// TwinCAT 3 PLC project PLC1
// ProgramVersion: 3.1.4026.24
// CompilerDefines: VISU_USEPROPERTYINFO
// libraries:
//   Tc2_Standard, * (Beckhoff Automation GmbH)
//   Tc2_System, * (Beckhoff Automation GmbH)
// project tree:
//   DUTs/ E_AutoStep.TcDUT, E_ControlMode.TcDUT (not stored), E_LogSev.TcDUT (not stored), E_MasterAutoStep.TcDUT, E_RobotConnState.TcDUT (not stored), ST_HmiMasterAuto.TcDUT, ST_HmiMasterAutoCfg.TcDUT, ST_HmiPiston.TcDUT, ST_HmiPistonAuto.TcDUT (not stored), ST_HmiPistonAutoCfg.TcDUT, ST_HmiRobot.TcDUT, ST_LogBridgeCfg.TcDUT (not stored), ST_LogEntry.TcDUT (not stored)
//   / GlobalTextList.TcGTLO, IOmapTask.TcTTO (not stored), PlcTask.TcTTO, Visualization Manager.TcVMO (not stored)
//   GVLs/ GVL_App.TcGVL, GVL_HMI.TcGVL, GVL_HmiPersistent.TcGVL, GVL_IO.TcGVL, GVL_Log.TcGVL, GVL_Robot.TcGVL (not stored)
//   POUs/ F_LogEvent.TcPOU, FB_MasterAutoCycle.TcPOU, FB_PistonAutoCycle.TcPOU, FB_SolSolPiston_2Pos.TcPOU, FB_SolSpringPiston_2Pos.TcPOU, MAIN.TcPOU, PRG_IoMap.TcPOU
//   VISUs/ VISU_Home.TcVIS, VISU_Piston.TcVIS, VISU_Pistons.TcVIS, VISU_Robot.TcVIS, VISU_AutoCycle.TcVIS, VISU_Diagnostics.TcVIS
// real-time tasks:
//   TASK PlcTask: cycle T#10ms, priority 20, ADS port 350
//   TASK IOmapTask: cycle T#5ms, priority 15, ADS port 351
// I/O:
//   DEVICE Device 1 (EtherCAT) (disabled), AmsNetId 192.168.1.101.2.1
//     Term 1 (EK1100) [EK1100 EtherCAT Coupler (2A E-Bus)]
//       Term 2 (EL2008) [EL2008 8Ch. Dig. Output 24V, 0.5A]
//       Term 3 (EL1008) [EL1008 8Ch. Dig. Input 24V, 3ms]
// variable links:
//   PLC1/PLC1 Instance <-> Device 1 (EtherCAT)/Term 1 (EK1100)/Term 2 (EL2008)
//     IOmapTask Outputs/GVL_IO.dOut[{1..8}] <-> Channel {1..8}/GVL_IO.dOut[{1..8}]  (8 links)
//   PLC1/PLC1 Instance <-> Device 1 (EtherCAT)/Term 1 (EK1100)/Term 3 (EL1008)
//     IOmapTask Inputs/GVL_IO.dIn[{1..8}] <-> Channel {1..8}/GVL_IO.dIn[{1..8}]  (8 links)

CONFIGURATION PLC1
    RESOURCE PLC ON TwinCAT3
        TASK PlcTask(INTERVAL := T#10ms, PRIORITY := 20);
        PROGRAM MAIN WITH PlcTask : MAIN;
    END_RESOURCE
END_CONFIGURATION

// ---- DUTs/E_AutoStep.TcDUT
{attribute 'qualified_only'}
{attribute 'strict'}
{attribute 'to_string'}
TYPE E_AutoStep :
(
    IDLE       := 0,
    EXTENDING  := 1,
    DWELL_EXT  := 2,
    RETRACTING := 3,
    DWELL_RET  := 4,
    ERR        := 99
) ;
END_TYPE

// ---- DUTs/E_MasterAutoStep.TcDUT
{attribute 'qualified_only'}
{attribute 'strict'}
{attribute 'to_string'}
TYPE E_MasterAutoStep :
(
    IDLE                 := 0,
    SEP_EXTENDING        := 1,
    WAIT_POS2            := 2,
    PUSH_EXTENDING       := 3,
    DWELL_PUSH           := 4,
    PUSH_RETRACTING      := 5,
    PUSH_RETRACTED_DWELL := 6,
    SEP_RETRACTING       := 7,
    SEP_RETRACTED_DWELL  := 8,
    INIT_PUSH_RETRACTING := 10,
    INIT_SEP_RETRACTING  := 11,
    INIT_GRIP_RETRACTING := 12,
    WAIT_PLATE           := 20,
    GRIP_EXTENDING       := 21,
    GRIP_RETRACTING      := 22,
    ERR                  := 99
) ;
END_TYPE

// ---- DUTs/ST_HmiMasterAuto.TcDUT
TYPE ST_HmiMasterAuto :
STRUCT
    // Display label ('MasterAuto'). Set from GVL_HMI init, never written by FB.
    Name             : STRING(30);

    // HMI writes -- momentary command buttons (R_TRIG inside FB latches the rising edge)
    bStart           : BOOL;
    bStop            : BOOL;
    bReset           : BOOL;

    // FB writes -- status
    eStep            : E_MasterAutoStep;
    sStepText        : STRING(20);   // human-readable mirror of eStep
    tElapsedS        : LREAL;        // seconds spent in the current step (0.0 on transition)
    iErrorCode       : INT;          // 0 = OK; see FB_MasterAutoCycle header for the code table
    sErrorText       : STRING(80);
    nCyclesCompleted : UDINT;        // incremented at end of GRIP_RETRACTING

    // HMI writes -- bench sim of the robot's start handshake. OR-ed with the
    // real stRobot.bStartAssembly level; FB auto-clears it after the rising
    // edge is consumed (never writes the robot-owned signal itself).
    bSimStartAssembly      : BOOL;

    // HMI writes -- per-step Simulate flags. Rising edge shortcuts the current
    // step's wait condition (FB clears the flag on consumption via R_TRIG.Q).
    bSimStep_Idle          : BOOL;
    bSimStep_InitPushRet   : BOOL;
    bSimStep_InitSepRet    : BOOL;
    bSimStep_InitGripRet   : BOOL;
    bSimStep_WaitPlate     : BOOL;
    bSimStep_GripExt       : BOOL;
    bSimStep_SepExt        : BOOL;
    bSimStep_WaitPos2      : BOOL;
    bSimStep_PushExt       : BOOL;
    bSimStep_DwellPush     : BOOL;
    bSimStep_PushRet       : BOOL;
    bSimStep_PushRetDwell  : BOOL;
    bSimStep_SepRet        : BOOL;
    bSimStep_SepRetDwell   : BOOL;
    bSimStep_GripRet       : BOOL;
END_STRUCT
END_TYPE

// ---- DUTs/ST_HmiMasterAutoCfg.TcDUT
TYPE ST_HmiMasterAutoCfg :
STRUCT
    // Timers, milliseconds. UDINT so HMI NumericInput binds directly.
    tDwellPushMs            : UDINT := 2000;   // DWELL_PUSH -- hold at push-extended
    tPushRetractedDwellMs   : UDINT := 500;    // PUSH_RETRACTED_DWELL -- hold after push retract
    tSepRetractedDwellMs    : UDINT := 500;    // SEP_RETRACTED_DWELL -- hold after sep retract before IDLE

    // Timeout guards every non-DWELL waiting state. On expiry, iErrorCode is
    // set to the step's numeric code and the cycle enters ERR.
    tStepTimeoutMs          : UDINT := 10000;

    // Dedicated timeout for WAIT_PLATE (bounded by robot placement time, not
    // by a motion budget). On expiry, iErrorCode := 9 and the cycle enters ERR.
    tPlateWaitTimeoutMs     : UDINT := 10000;

    // If TRUE, the 4 movement states ignore sensor feedback and advance when
    // tStepTimeoutMs expires — the timeout doubles as the fixed step duration.
    // No timeout-error path while sensorless. Mirrors ST_HmiPistonAutoCfg.bNoSensors.
    bNoSensors              : BOOL  := FALSE;

    // While TRUE, IDLE immediately starts the next cycle (no START or
    // robot CMD:1 edge needed). Uncheck to stop after the cycle returns
    // to IDLE. Cleared by the FB on entry to ERR so a RESET does not
    // instantly restart motion.
    bContinuous             : BOOL  := FALSE;

    // Global machine mode — single source of truth for every piston's mode.
    // BOOL so the classic VISU HMI (boolean-only) binds a checkbox directly,
    // matching the per-piston bMode convention. FALSE = Manual (operator jogs
    // each piston; master cycle held in IDLE). TRUE = Automatic (MasterAutoCycle
    // owns all six pistons). Enforced every scan in MAIN onto each piston's
    // eMode AND bMode, so there is no per-piston double-control.
    bAutoMode               : BOOL := FALSE;
END_STRUCT
END_TYPE

// ---- DUTs/ST_HmiPiston.TcDUT
TYPE ST_HmiPiston :
STRUCT
    // Display label ("Piston 1", "Ejector", ...). Set from GVL_HMI, never written by FB.
    Name               : STRING(30);

    // HMI writes — mode
    eMode              : E_ControlMode;
	bMode				: BOOL; // to be able to control from the VISU old HMI

    // HMI writes — latched command targets (momentary press, rising edge selects)
    bManCmdExtend      : BOOL;
    bManCmdRetract     : BOOL;

    // HMI writes — jog while held (TRUE while operator holds the JOG button)
    bManJogExtend      : BOOL;
    bManJogRetract     : BOOL;

    // HMI writes — simulate sensor inputs (OR-merged with real). Future Sim checkbox hook.
    bSimulateExtended  : BOOL;
    bSimulateRetracted : BOOL;

    // HMI reads (FB writes) — latched-target highlight
    bSelectedExtend    : BOOL;
    bSelectedRetract   : BOOL;

    // HMI reads (FB writes) — effective sensor = real OR simulate
    bIsExtended        : BOOL;
    bIsRetracted       : BOOL;
    bIsMoving          : BOOL;

    // HMI reads — physical solenoid coil states (FB mirrors them every cycle)
    bOutSolenoidExtend  : BOOL;
    bOutSolenoidRetract : BOOL;
END_STRUCT
END_TYPE

// ---- DUTs/ST_HmiPistonAutoCfg.TcDUT
TYPE ST_HmiPistonAutoCfg :
STRUCT
    // All times in milliseconds. UDINT so HMI NumericInput binds directly (no TIME<->UDINT juggling).

    // Dwell = how long to sit at the sensor before starting the reverse move.
    tDwellExtendedMs   : UDINT := 500;
    tDwellRetractedMs  : UDINT := 500;

    // Timeout = if we do not see the target sensor within this window, raise an error.
    tTimeoutExtendMs   : UDINT := 3000;
    tTimeoutRetractMs  : UDINT := 3000;

    // If TRUE, DWELL_RET loops back to EXTENDING instead of returning to IDLE.
    bContinuous        : BOOL  := FALSE;
END_STRUCT
END_TYPE

// ---- DUTs/ST_HmiRobot.TcDUT
TYPE ST_HmiRobot :
STRUCT
    // Display label ('Robot'). Set from GVL_Robot, never written by bridge.
    Name           : STRING(30);

    // Bridge writes — connection state (enum + string mirror for HMI text binding)
    eConnState     : E_RobotConnState;
    sConnStateText : STRING(20);

    // Bridge writes — latched "in position N" flags. Bridge holds the last-seen
    // position TRUE and clears the other two when a new POS frame arrives.
    bAtPos1        : BOOL;
    bAtPos2        : BOOL;
    bAtPos3        : BOOL;

    // Bridge writes — diagnostics
    nPacketsRx     : UDINT;
    sLastMessage   : STRING(80);

    // Outbound pulses — PLC (FB_MasterAutoCycle) writes TRUE for one cycle.
    // Bridge polls each on rising edge, sends the corresponding TCP frame,
    // then clears the flag. If the bridge is disconnected the flag stays
    // TRUE until reconnect; no queue, no lost pulses.
    bTxAutoStarted  : BOOL;
    bTxPushDone     : BOOL;
    bTxPistonsError : BOOL;

    // Inbound pulse — bridge writes TRUE on receiving a RESET_ERROR frame.
    // FB_MasterAutoCycle consumes on rising edge and clears the flag.
    bRxResetError   : BOOL;

    // Bridge writes — outbound diagnostics
    nPacketsTx      : UDINT;
    sLastTxMessage  : STRING(80);
END_STRUCT
END_TYPE

// ---- GVLs/GVL_App.TcGVL
{attribute 'qualified_only'}
// Cooked IO aliases. Bound to the raw GVL_IO.dIn[i]/dOut[i] hardware arrays
// in MAIN's read-inputs / write-outputs bookends. No AT %*: these are plain
// BOOLs the FBs consume — the actual hardware wiring lives in GVL_IO.
//
// Tag convention: <Device>Sol<N>  = single EXTEND coil (SOL-Spring).
// The mechanical spring returns the actuator when the coil is de-energised,
// so no per-actuator Retract alias exists. DI still has a Retracted sensor.
//
//   SepSolN : Pin separator N   (DI 1..6, DO 1..3)
//   PushSolN: Pin push N        (DI 7..12, DO 4..6)
//   GripSolL / GripSolR: side grip pistons that clamp the robot-placed plate
//                       (DI 14..17, DO 8..9)
//   PlateSenL / PlateSenR: plate-presence sensors gating cycle start
//                         (DI 18..19)
//   PbN / LedPbN: panel push buttons + status LEDs (DI 20..22, DO 10..12).
//                Behavior mode-gated -- see field comments below.
//
// DO layout:
//   dOut[1..3] = SepSolN Extend
//   dOut[4..6] = PushSolN Extend
//   dOut[7]    = free (was Robot bAssemblyRunning; retired, comms are TCP-only)
//   dOut[8..9] = GripSolL/R Extend
//   dOut[10..12] = PB1/2/3 LEDs (see Phase B)
//   dOut[13..16] = free
VAR_GLOBAL
    // SepSol1 (Pin separator 1) — DI 1..2, DO 1
    bSensorSepRetracted1  : BOOL;
    bSensorSepExtended1   : BOOL;
    bValveSepExtend1      : BOOL;

    // SepSol2 (Pin separator 2) — DI 3..4, DO 2
    bSensorSepRetracted2  : BOOL;
    bSensorSepExtended2   : BOOL;
    bValveSepExtend2      : BOOL;

    // SepSol3 (Pin separator 3) — DI 5..6, DO 3
    bSensorSepRetracted3  : BOOL;
    bSensorSepExtended3   : BOOL;
    bValveSepExtend3      : BOOL;

    // PushSol1 (Pin push 1) — DI 7..8, DO 4
    bSensorPushRetracted1 : BOOL;
    bSensorPushExtended1  : BOOL;
    bValvePushExtend1     : BOOL;

    // PushSol2 (Pin push 2) — DI 9..10, DO 5
    bSensorPushRetracted2 : BOOL;
    bSensorPushExtended2  : BOOL;
    bValvePushExtend2     : BOOL;

    // PushSol3 (Pin push 3) — DI 11..12, DO 6
    bSensorPushRetracted3 : BOOL;
    bSensorPushExtended3  : BOOL;
    bValvePushExtend3     : BOOL;

    // GripSolL (side grip, left) — DI 14..15, DO 8
    bSensorGripRetractedL : BOOL;
    bSensorGripExtendedL  : BOOL;
    bValveGripExtendL     : BOOL;

    // GripSolR (side grip, right) — DI 16..17, DO 9
    bSensorGripRetractedR : BOOL;
    bSensorGripExtendedR  : BOOL;
    bValveGripExtendR     : BOOL;

    // Plate-presence sensors — DI 18..19 (input only; no coil)
    bPlateSenL : BOOL;
    bPlateSenR : BOOL;

    // Panel push buttons + status LEDs — DI 20..22 / DO 10..12.
    // PB1 in Auto  = cycle-start bypass (bypass of robot's CMD:1).
    // PB1 in Manual = hold to extend both grip pistons.
    // PB2 in Manual = hold to extend all 3 SepSol pistons.
    // PB3 in Manual = hold to extend all 3 PushSol pistons.
    // LEDs mirror the corresponding PB press state (wiring diagnostic).
    bPb1     : BOOL;
    bPb2     : BOOL;
    bPb3     : BOOL;
    bLedPb1  : BOOL;
    bLedPb2  : BOOL;
    bLedPb3  : BOOL;
END_VAR

// ---- GVLs/GVL_HMI.TcGVL
{attribute 'qualified_only'}
{attribute 'TcHmiSymbol.AddSymbol'}
VAR_GLOBAL
    stSepSol1  : ST_HmiPiston := (Name := 'SepSol1');
    stSepSol2  : ST_HmiPiston := (Name := 'SepSol2');
    stSepSol3  : ST_HmiPiston := (Name := 'SepSol3');
    stPushSol1 : ST_HmiPiston := (Name := 'PushSol1');
    stPushSol2 : ST_HmiPiston := (Name := 'PushSol2');
    stPushSol3 : ST_HmiPiston := (Name := 'PushSol3');
    stGripSolL : ST_HmiPiston := (Name := 'GripSolL');
    stGripSolR : ST_HmiPiston := (Name := 'GripSolR');

    // Runtime state for the per-piston auto sequencers. Config for each
    // lives in the matching stXxxAutoCfg in GVL_HmiPersistent (PERSISTENT).
    stSepSol1Auto  : ST_HmiPistonAuto;
    stSepSol2Auto  : ST_HmiPistonAuto;
    stSepSol3Auto  : ST_HmiPistonAuto;
    stPushSol1Auto : ST_HmiPistonAuto;
    stPushSol2Auto : ST_HmiPistonAuto;
    stPushSol3Auto : ST_HmiPistonAuto;

    // Plate-presence sensors exposed to the HMI (indicator lamps on the
    // AutoCycle page). Mirror of GVL_App.bPlateSen* driven in MAIN.
    bPlateSenL : BOOL;
    bPlateSenR : BOOL;

    // Runtime state for the master (multi-piston + robot-coordinated) auto
    // sequence. Config for it lives in GVL_HmiPersistent.stMasterAutoCfg.
    stMasterAuto   : ST_HmiMasterAuto := (Name := 'MasterAuto');
END_VAR

// ---- GVLs/GVL_HmiPersistent.TcGVL
{attribute 'qualified_only'}
{attribute 'TcHmiSymbol.AddSymbol'}
VAR_GLOBAL PERSISTENT
    // Auto-cycle configuration. PERSISTENT so operator-tuned dwell / timeout
    // values survive an Activate Configuration + PLC restart. Values reset
    // to the struct defaults only on a full cold-boot reset.
    stSepSol1AutoCfg  : ST_HmiPistonAutoCfg;
    stPushSol1AutoCfg : ST_HmiPistonAutoCfg;

    // Config for the master (multi-piston + robot-coordinated) auto sequence.
    // See ST_HmiMasterAutoCfg for the tunable list; defaults land on cold-boot.
    stMasterAutoCfg   : ST_HmiMasterAutoCfg;
END_VAR

// ---- GVLs/GVL_IO.TcGVL
{attribute 'qualified_only'}
VAR_GLOBAL
	dOut AT%Q* :ARRAY[1..16]OF BOOL;
	dIn  AT%I* :ARRAY[1..24]OF BOOL;
END_VAR

// ---- GVLs/GVL_Log.TcGVL
{attribute 'qualified_only'}
{attribute 'TcHmiSymbol.AddSymbol'}
VAR_GLOBAL
    // Ring buffer of the most recent log entries the PLC has produced.
    // The Python bridge polls nWriteIdx via ADS and drains new slots.
    //   write slot at any moment = (nWriteIdx MOD 256)
    //   overflow detected when (nWriteIdx - lastReadIdx) > 256
    aLog       : ARRAY[0..255] OF ST_LogEntry;

    // Monotonic write counter (never wraps in practice — UDINT overflows
    // after 2^32 writes ≈ 4.3 billion, decades even at 1 kHz logging).
    nWriteIdx  : UDINT;

    // Runtime toggle for DEBUG severity. F_LogEvent drops DBG entries
    // when this is FALSE. Operator can flip it from the HMI without a
    // rebuild. HMI ToggleSwitch on the Robot page binds here.
    bDebugMode : BOOL := FALSE;
END_VAR

// ---- POUs/MAIN.TcPOU
PROGRAM MAIN
VAR
    fbSepSol1  : FB_SolSpringPiston_2Pos;
    fbSepSol2  : FB_SolSpringPiston_2Pos;
    fbSepSol3  : FB_SolSpringPiston_2Pos;
    fbPushSol1 : FB_SolSpringPiston_2Pos;
    fbPushSol2 : FB_SolSpringPiston_2Pos;
    fbPushSol3 : FB_SolSpringPiston_2Pos;

    // Per-piston auto-cycle sequencers. Each drives one piston's
    // bAutoCmdExtend / bAutoCmdRetract via its bCmdExtend / bCmdRetract,
    // OR-merged with fbMasterAutoCycle's output at each piston call site.
    fbSepSol1Auto  : FB_PistonAutoCycle;
    fbSepSol2Auto  : FB_PistonAutoCycle;
    fbSepSol3Auto  : FB_PistonAutoCycle;
    fbPushSol1Auto : FB_PistonAutoCycle;
    fbPushSol2Auto : FB_PistonAutoCycle;
    fbPushSol3Auto : FB_PistonAutoCycle;

    // Full-machine sequencer coordinating the 3 pairs of (SepSolN,
    // PushSolN) plus the robot handshake. Its command outputs
    // OR-merge with the per-piston auto FBs at each piston call site.
    fbMasterAutoCycle : FB_MasterAutoCycle;
END_VAR

(* ==========================================
   Master auto-cycle — coordinates the 3 pairs of (Sep,Push) pistons
   with the robot handshake. Called BEFORE the per-piston
   auto FBs and BEFORE the piston FBs so its bSepCmd* / bPushCmd*
   outputs feed forward this scan.
   Master reads bIs* from the piston stHmi structs — those carry the
   previous scan's values (100 µs lag, negligible for a physical
   machine).
   ========================================== *)
fbMasterAutoCycle.bSepIsExtended[1]   := GVL_HMI.stSepSol1.bIsExtended;
fbMasterAutoCycle.bSepIsExtended[2]   := GVL_HMI.stSepSol2.bIsExtended;
fbMasterAutoCycle.bSepIsExtended[3]   := GVL_HMI.stSepSol3.bIsExtended;
fbMasterAutoCycle.bSepIsRetracted[1]  := GVL_HMI.stSepSol1.bIsRetracted;
fbMasterAutoCycle.bSepIsRetracted[2]  := GVL_HMI.stSepSol2.bIsRetracted;
fbMasterAutoCycle.bSepIsRetracted[3]  := GVL_HMI.stSepSol3.bIsRetracted;
fbMasterAutoCycle.bPushIsExtended[1]  := GVL_HMI.stPushSol1.bIsExtended;
fbMasterAutoCycle.bPushIsExtended[2]  := GVL_HMI.stPushSol2.bIsExtended;
fbMasterAutoCycle.bPushIsExtended[3]  := GVL_HMI.stPushSol3.bIsExtended;
fbMasterAutoCycle.bPushIsRetracted[1] := GVL_HMI.stPushSol1.bIsRetracted;
fbMasterAutoCycle.bPushIsRetracted[2] := GVL_HMI.stPushSol2.bIsRetracted;
fbMasterAutoCycle.bPushIsRetracted[3] := GVL_HMI.stPushSol3.bIsRetracted;
fbMasterAutoCycle(
    bStartAssembly := GVL_Robot.stRobot.bStartAssembly,
    stHmi          := GVL_HMI.stMasterAuto,
    stCfg          := GVL_HmiPersistent.stMasterAutoCfg,
    stRobot        := GVL_Robot.stRobot
);

(* Optional "Put all to Auto" mode: while the master cycle is running,
   force all six pistons into Automatic so bAutoCmd* reaches the coil.
   Gated by stMasterAutoCfg.bForceAllAuto — when FALSE (default), only
   pistons the operator explicitly put into Automatic participate in the
   master cycle. On IDLE / ERR this block does nothing, regardless of
   the flag. *)
IF fbMasterAutoCycle.bAnyRunning AND GVL_HmiPersistent.stMasterAutoCfg.bForceAllAuto THEN
    GVL_HMI.stSepSol1.eMode  := E_ControlMode.Automatic;
    GVL_HMI.stPushSol1.eMode := E_ControlMode.Automatic;
    GVL_HMI.stSepSol2.eMode  := E_ControlMode.Automatic;
    GVL_HMI.stPushSol2.eMode := E_ControlMode.Automatic;
    GVL_HMI.stSepSol3.eMode  := E_ControlMode.Automatic;
    GVL_HMI.stPushSol3.eMode := E_ControlMode.Automatic;
END_IF;

(* ==========================================
   Pin separators (SOL-Spring, 2 limit switches, single Extend coil).
   SepSol1 and PushSol1 are driven by their own FB_PistonAutoCycle
   instances (called first so their outputs feed the piston FB this
   cycle). All six pistons OR-merge with fbMasterAutoCycle's outputs
   so the master sequence can command any/all of them in parallel.
   ========================================== *)
fbSepSol1Auto(
    sName        := 'SepSol1Auto',
    stHmi        := GVL_HMI.stSepSol1,
    stAuto       := GVL_HMI.stSepSol1Auto,
    stCfg        := GVL_HmiPersistent.stSepSol1AutoCfg
    // bCmdExtend / bCmdRetract wired inline in the fbSepSol1 call below
);

fbSepSol1(
    bAutoCmdExtend   := fbSepSol1Auto.bCmdExtend  OR fbMasterAutoCycle.bSepCmdExtend[1],
    bAutoCmdRetract  := fbSepSol1Auto.bCmdRetract OR fbMasterAutoCycle.bSepCmdRetract[1],
    bSwitchExtended  := GVL_App.bSensorSepExtended1,
    bSwitchRetracted := GVL_App.bSensorSepRetracted1,
    stHmi            := GVL_HMI.stSepSol1,
    bOutSolenoid     => GVL_App.bValveSepExtend1
);

fbSepSol2Auto(
    sName        := 'SepSol2Auto',
    stHmi        := GVL_HMI.stSepSol2,
    stAuto       := GVL_HMI.stSepSol2Auto,
    stCfg        := GVL_HmiPersistent.stSepSol2AutoCfg
);

fbSepSol2(
    bAutoCmdExtend   := fbSepSol2Auto.bCmdExtend  OR fbMasterAutoCycle.bSepCmdExtend[2],
    bAutoCmdRetract  := fbSepSol2Auto.bCmdRetract OR fbMasterAutoCycle.bSepCmdRetract[2],
    bSwitchExtended  := GVL_App.bSensorSepExtended2,
    bSwitchRetracted := GVL_App.bSensorSepRetracted2,
    stHmi            := GVL_HMI.stSepSol2,
    bOutSolenoid     => GVL_App.bValveSepExtend2
);

fbSepSol3Auto(
    sName        := 'SepSol3Auto',
    stHmi        := GVL_HMI.stSepSol3,
    stAuto       := GVL_HMI.stSepSol3Auto,
    stCfg        := GVL_HmiPersistent.stSepSol3AutoCfg
);

fbSepSol3(
    bAutoCmdExtend   := fbSepSol3Auto.bCmdExtend  OR fbMasterAutoCycle.bSepCmdExtend[3],
    bAutoCmdRetract  := fbSepSol3Auto.bCmdRetract OR fbMasterAutoCycle.bSepCmdRetract[3],
    bSwitchExtended  := GVL_App.bSensorSepExtended3,
    bSwitchRetracted := GVL_App.bSensorSepRetracted3,
    stHmi            := GVL_HMI.stSepSol3,
    bOutSolenoid     => GVL_App.bValveSepExtend3
);

(* ==========================================
   Pin pushers
   ========================================== *)
fbPushSol1Auto(
    sName        := 'PushSol1Auto',
    stHmi        := GVL_HMI.stPushSol1,
    stAuto       := GVL_HMI.stPushSol1Auto,
    stCfg        := GVL_HmiPersistent.stPushSol1AutoCfg
    // bCmdExtend / bCmdRetract wired inline in the fbPushSol1 call below
);

fbPushSol1(
    bAutoCmdExtend   := fbPushSol1Auto.bCmdExtend  OR fbMasterAutoCycle.bPushCmdExtend[1],
    bAutoCmdRetract  := fbPushSol1Auto.bCmdRetract OR fbMasterAutoCycle.bPushCmdRetract[1],
    bSwitchExtended  := GVL_App.bSensorPushExtended1,
    bSwitchRetracted := GVL_App.bSensorPushRetracted1,
    stHmi            := GVL_HMI.stPushSol1,
    bOutSolenoid     => GVL_App.bValvePushExtend1
);

fbPushSol2Auto(
    sName        := 'PushSol2Auto',
    stHmi        := GVL_HMI.stPushSol2,
    stAuto       := GVL_HMI.stPushSol2Auto,
    stCfg        := GVL_HmiPersistent.stPushSol2AutoCfg
);

fbPushSol2(
    bAutoCmdExtend   := fbPushSol2Auto.bCmdExtend  OR fbMasterAutoCycle.bPushCmdExtend[2],
    bAutoCmdRetract  := fbPushSol2Auto.bCmdRetract OR fbMasterAutoCycle.bPushCmdRetract[2],
    bSwitchExtended  := GVL_App.bSensorPushExtended2,
    bSwitchRetracted := GVL_App.bSensorPushRetracted2,
    stHmi            := GVL_HMI.stPushSol2,
    bOutSolenoid     => GVL_App.bValvePushExtend2
);

fbPushSol3Auto(
    sName        := 'PushSol3Auto',
    stHmi        := GVL_HMI.stPushSol3,
    stAuto       := GVL_HMI.stPushSol3Auto,
    stCfg        := GVL_HmiPersistent.stPushSol3AutoCfg
);

fbPushSol3(
    bAutoCmdExtend   := fbPushSol3Auto.bCmdExtend  OR fbMasterAutoCycle.bPushCmdExtend[3],
    bAutoCmdRetract  := fbPushSol3Auto.bCmdRetract OR fbMasterAutoCycle.bPushCmdRetract[3],
    bSwitchExtended  := GVL_App.bSensorPushExtended3,
    bSwitchRetracted := GVL_App.bSensorPushRetracted3,
    stHmi            := GVL_HMI.stPushSol3,
    bOutSolenoid     => GVL_App.bValvePushExtend3
);

END_PROGRAM

// ---- POUs/FB_SolSpringPiston_2Pos.TcPOU
FUNCTION_BLOCK FB_SolSpringPiston_2Pos
(* Single-solenoid, spring-return 2-position actuator.
   Coil energised  -> drives to EXTENDED.
   Coil de-energised -> mechanical spring returns to RETRACTED.

   The coil is a continuous force against the spring, so Section 2 uses a
   LATCH-and-RETAIN pattern: the coil is set TRUE on Extend command and
   FALSE on Retract command, and RETAINS its state (via VAR_OUTPUT retain)
   any cycle no explicit command is active. Without the latch the coil
   would drop the moment the extended sensor fires and the spring would
   immediately pull the piston back.

   Fail-safe by construction: broken wire, dead coil, PLC power loss
   or e-stop all leave bOutSolenoid FALSE and the spring retracts.

   Interface is kept symmetric with FB_SolSolPiston_2Pos so a sequencer FB
   (e.g. FB_PistonAutoCycle) can drive either actuator type without a
   custom variant. Reuses ST_HmiPiston unchanged; the retract-coil mirror
   field (stHmi.bOutSolenoidRetract) is always FALSE because no retract
   coil exists on this actuator. *)
VAR_INPUT
    (* Automatic Commands from PLC sequence logic. Wired to FALSE in MAIN until FB_Auto exists. *)
    bAutoCmdExtend    : BOOL;
    bAutoCmdRetract   : BOOL;

    (* External jog request (e.g. panel push-button). OR-merged with the
       HMI's stHmi.bManJogExtend inside so a physical PB and the HMI
       button can drive the same jog without stepping on each other.
       Only takes effect while eMode = Manual (same gate as the HMI jog). *)
    bJogExtend        : BOOL;

    (* Physical Feedback (Proximity Switches) *)
    bSwitchExtended   : BOOL;
    bSwitchRetracted  : BOOL;
END_VAR

VAR_IN_OUT
    (* HMI contract — mode, manual + simulate inputs, latched + sensor status *)
    stHmi             : ST_HmiPiston;
END_VAR

VAR_OUTPUT
    (* Physical Output to Solenoid — SINGLE coil.
       TRUE  = coil energised, actuator drives EXTENDED.
       FALSE = coil de-energised, spring returns actuator to RETRACTED. *)
    bOutSolenoid      : BOOL;
END_VAR

VAR
    (* Internal Target States *)
    bTargetExtend     : BOOL;
    bTargetRetract    : BOOL;

    (* HMI Manual-Button Edge Detection *)
    fbTrigManExtend   : R_TRIG;
    fbTrigManRetract  : R_TRIG;

    (* Effective sensor states = real OR HMI simulate. Recomputed every cycle in Section 0a. *)
    bSwitchExtended_eff  : BOOL;
    bSwitchRetracted_eff : BOOL;

    (* Previous-cycle snapshots for the mode-field bridge in Section 0b.
       Classic PLC HMI writes stHmi.bMode (Rotary Switch is boolean-only);
       web HMI writes stHmi.eMode (enum via ToggleSwitch). This FB is the
       authoritative reader of eMode, so we sync in whichever direction
       changed since last cycle. *)
    bPrevMode : BOOL;
    ePrevMode : E_ControlMode;
END_VAR

(* ==========================================
   0b. MODE-FIELD BRIDGE — sync bMode <-> eMode
   The classic PLC HMI (VISUs) writes stHmi.bMode because its Rotary Switch
   element is boolean-only. The web HMI (Flower_HMI) writes stHmi.eMode via
   a ToggleSwitch. Rest of this FB reads eMode as the authoritative field,
   so we mirror bMode into eMode when the classic HMI toggled the switch,
   and mirror eMode back into bMode when the web HMI (or anyone else) wrote
   eMode. Edge-triggered — whichever side changed since last cycle wins.
   Runs BEFORE Section 0 so downstream logic sees a coherent eMode.
   ========================================== *)
IF stHmi.bMode <> bPrevMode THEN
    // Classic VISU changed bMode → propagate to eMode
    IF stHmi.bMode THEN
        stHmi.eMode := E_ControlMode.Automatic;
    ELSE
        stHmi.eMode := E_ControlMode.Manual;
    END_IF;
ELSIF stHmi.eMode <> ePrevMode THEN
    // Web HMI (or any other writer) changed eMode → propagate to bMode
    stHmi.bMode := (stHmi.eMode = E_ControlMode.Automatic);
END_IF;

bPrevMode := stHmi.bMode;
ePrevMode := stHmi.eMode;

(* ==========================================
   0a. EFFECTIVE SENSOR INPUTS (real OR HMI simulate)
   ========================================== *)
bSwitchExtended_eff  := bSwitchExtended  OR stHmi.bSimulateExtended;
bSwitchRetracted_eff := bSwitchRetracted OR stHmi.bSimulateRetracted;

(* ==========================================
   0. HMI MANUAL BUTTON LATCHING (Radio-Button Behavior)
   ========================================== *)
fbTrigManExtend(CLK := stHmi.bManCmdExtend);
fbTrigManRetract(CLK := stHmi.bManCmdRetract);

// Independent IFs (not ELSIF): if multiple edges fire in the same cycle, the last one wins (Retract > Extend).
IF fbTrigManExtend.Q  THEN stHmi.bSelectedExtend := TRUE;  stHmi.bSelectedRetract := FALSE; END_IF;
IF fbTrigManRetract.Q THEN stHmi.bSelectedExtend := FALSE; stHmi.bSelectedRetract := TRUE;  END_IF;

IF stHmi.eMode = E_ControlMode.Automatic THEN
    stHmi.bSelectedExtend := FALSE; stHmi.bSelectedRetract := FALSE;
END_IF;

(* ==========================================
   1. MODE SELECTION & COMMAND MAPPING
   Spring-return semantics: both bAutoCmd* inputs are accepted for interface
   parity with FB_SolSolPiston_2Pos, but physically only Extend commands the
   coil. If both auto bits are TRUE we treat it as a conflict and de-energise
   (safe default — spring retracts).
   ========================================== *)
IF stHmi.eMode = E_ControlMode.Automatic THEN
    bTargetExtend  := bAutoCmdExtend  AND NOT bAutoCmdRetract;
    bTargetRetract := bAutoCmdRetract AND NOT bAutoCmdExtend;

ELSIF stHmi.eMode = E_ControlMode.Manual THEN
    bTargetExtend  := stHmi.bSelectedExtend;
    bTargetRetract := stHmi.bSelectedRetract;

ELSE
    // Safe default: undefined mode → no targets
    bTargetExtend  := FALSE;
    bTargetRetract := FALSE;
END_IF;

(* ==========================================
   1a. JOG OVERRIDE — clear latched selection while either jog is held
   ========================================== *)
// Section 1 above already copied stHmi.bSelected* into bTarget*. The stale
// bTarget* is harmless because Section 2's jog branches sit ahead of the
// bTarget* branches in the IF/ELSIF ladder and preempt them.
IF stHmi.bManJogExtend OR stHmi.bManJogRetract OR bJogExtend THEN
    stHmi.bSelectedExtend := FALSE; stHmi.bSelectedRetract := FALSE;
END_IF;

(* ==========================================
   1b. TARGET-REACHED RESET — clear bSelected* once the piston arrives
   ========================================== *)
IF stHmi.bSelectedExtend  AND bSwitchExtended_eff  THEN stHmi.bSelectedExtend  := FALSE; END_IF;
IF stHmi.bSelectedRetract AND bSwitchRetracted_eff THEN stHmi.bSelectedRetract := FALSE; END_IF;

(* ==========================================
   2. SOLENOID CONTROL — single coil, LATCH-and-RETAIN
   The coil is a continuous force against the spring. If it drops, the spring
   wins and the actuator retracts. So the coil must be LATCHED TRUE from the
   moment Extend is commanded until Retract is commanded — not pulsed until
   the sensor fires (which is the double-solenoid pattern).
   Structure:
     - Jog branches first, gated by Manual mode.
     - Explicit Extend / Retract command branches drive the coil to a
       definite state.
     - The IF ladder has NO ELSE. When no branch matches, VAR_OUTPUT retain
       semantics carry the coil forward:
         * At the Extended sensor after a successful extend (Section 1b just
           cleared bTargetExtend) → coil retains TRUE → piston HOLDS.
         * At the Retracted sensor after a successful retract → coil retains
           FALSE → piston HOLDS retracted (spring already there).
         * Sequencer DWELL_EXT (both auto bits FALSE) → coil retains TRUE
           for the full dwell instead of releasing the piston.
     - No sensor guards on the drive branches: holding the coil TRUE while
       at the Extended sensor is normal operation, not a wasted drive.
   Fail-safe still holds: cold boot, PLC reset, or e-stop leave bOutSolenoid
   at its default FALSE and the spring retracts.
   ========================================== *)
// JOG EXTEND: while held in Manual, energise coil. HMI-owned bManJogExtend
// OR external bJogExtend (panel push-button) -- both share the Manual gate.
IF (stHmi.bManJogExtend OR bJogExtend) AND stHmi.eMode = E_ControlMode.Manual THEN
    bOutSolenoid := TRUE;

// JOG RETRACT: while held in Manual, de-energise coil (spring retracts)
ELSIF stHmi.bManJogRetract AND stHmi.eMode = E_ControlMode.Manual THEN
    bOutSolenoid := FALSE;

// EXTEND commanded — energise coil (latched via retain when bTargetExtend clears)
ELSIF bTargetExtend THEN
    bOutSolenoid := TRUE;

// RETRACT commanded — de-energise coil, spring retracts
ELSIF bTargetRetract THEN
    bOutSolenoid := FALSE;

// No branch → bOutSolenoid RETAINS its previous value (see block header).
END_IF;

(* ==========================================
   3. HMI STATUS FEEDBACK
   bIsMoving is derived from sensor state alone: with Section 2's latch
   semantics, bOutSolenoid stays TRUE at the extended limit — so ORing
   it in would report "moving" while the piston is actually parked.
   "Between the two limits" is accurate for both strokes: coil-driven
   extend and spring-driven retract both traverse that gap.

   bOutSolenoidRetract is written FALSE unconditionally — no retract coil
   exists on a spring-return actuator, so the mirror stays cleared.
   ========================================== *)
stHmi.bIsExtended         := bSwitchExtended_eff;
stHmi.bIsRetracted        := bSwitchRetracted_eff;
stHmi.bIsMoving           := NOT bSwitchExtended_eff AND NOT bSwitchRetracted_eff;
stHmi.bOutSolenoidExtend  := bOutSolenoid;
stHmi.bOutSolenoidRetract := FALSE;

END_FUNCTION_BLOCK

// ---- POUs/FB_PistonAutoCycle.TcPOU
FUNCTION_BLOCK FB_PistonAutoCycle
VAR_INPUT
    (* Instance name used as the log source (e.g. 'SepSol1Auto').
       Kept as VAR_INPUT so the FB is reusable across pistons — MAIN passes
       the actual name at each call site. *)
    sName : STRING(20);
END_VAR

VAR_IN_OUT
    (* Reads bIs* effective sensors, writes eMode := Automatic while running. *)
    stHmi  : ST_HmiPiston;
    (* Reads commands, writes step + status. *)
    stAuto : ST_HmiPistonAuto;
    (* Reads persistent dwell / timeout / continuous config. *)
    stCfg  : ST_HmiPistonAutoCfg;
END_VAR

VAR_OUTPUT
    (* Wire these to the piston FB's bAutoCmdExtend / bAutoCmdRetract in MAIN. *)
    bCmdExtend  : BOOL;
    bCmdRetract : BOOL;
END_VAR

VAR
    (* HMI button edge detection *)
    fbTrigStart : R_TRIG;
    fbTrigStop  : R_TRIG;
    fbTrigReset : R_TRIG;
    fbTrigAck   : R_TRIG;

    (* Per-state timers. TON.IN bound to (eStep = target); .Q fires when PT elapsed.
       When we transition out, IN goes FALSE and TON auto-resets ET. *)
    fbTimerExtend  : TON;   // extend-timeout (fault on Q while EXTENDING)
    fbTimerRetract : TON;   // retract-timeout (fault on Q while RETRACTING)
    fbTimerDwellE  : TON;   // dwell at extended
    fbTimerDwellR  : TON;   // dwell at retracted

    (* Step-elapsed display timer. Resets on step change; long PT so .Q never fires. *)
    fbStepTimer : TON;

    (* Prev-state snapshot for step-changed detection *)
    ePrevStep    : E_AutoStep;
    bStepChanged : BOOL;
END_VAR

(* ==========================================
   0. HMI COMMAND EDGE DETECTION
   ========================================== *)
fbTrigStart(CLK := stAuto.bStart);
fbTrigStop (CLK := stAuto.bStop);
fbTrigReset(CLK := stAuto.bReset);
fbTrigAck  (CLK := stAuto.bAck);

(* ==========================================
   1. PER-STATE TIMERS
   Called BEFORE the state machine so their .Q outputs reflect the current
   state's dwell / timeout for this cycle's decisions.
   ========================================== *)
fbTimerExtend (IN := stAuto.eStep = E_AutoStep.EXTENDING,  PT := UDINT_TO_TIME(stCfg.tTimeoutExtendMs));
fbTimerRetract(IN := stAuto.eStep = E_AutoStep.RETRACTING, PT := UDINT_TO_TIME(stCfg.tTimeoutRetractMs));
fbTimerDwellE (IN := stAuto.eStep = E_AutoStep.DWELL_EXT,  PT := UDINT_TO_TIME(stCfg.tDwellExtendedMs));
fbTimerDwellR (IN := stAuto.eStep = E_AutoStep.DWELL_RET,  PT := UDINT_TO_TIME(stCfg.tDwellRetractedMs));

(* ==========================================
   2. GLOBAL COMMANDS
   Stop = soft interrupt back to IDLE (does NOT clear error latch).
   Reset = hard reset: force IDLE, clear cycles + error.
   Ack = clear error latch (only meaningful from ERR).
   ========================================== *)
IF fbTrigStop.Q AND stAuto.eStep <> E_AutoStep.ERR THEN
    stAuto.eStep := E_AutoStep.IDLE;
END_IF

IF fbTrigReset.Q THEN
    stAuto.eStep            := E_AutoStep.IDLE;
    stAuto.bError           := FALSE;
    stAuto.sErrorText       := '';
    stAuto.nCyclesCompleted := 0;
END_IF

IF fbTrigAck.Q AND stAuto.eStep = E_AutoStep.ERR THEN
    stAuto.bError     := FALSE;
    stAuto.sErrorText := '';
    stAuto.eStep      := E_AutoStep.IDLE;
END_IF

(* ==========================================
   3. STATE MACHINE
   Reads effective sensors from stHmi.bIsExtended / bIsRetracted — these
   are already the real-OR-simulate value written by the piston FB
   (FB_SolSolPiston_2Pos or FB_SolSpringPiston_2Pos). So simulation
   "just works" via the piston FB's existing bSimulate* pins.
   ========================================== *)
CASE stAuto.eStep OF

    E_AutoStep.IDLE:
        bCmdExtend  := FALSE;
        bCmdRetract := FALSE;
        (* Start only from IDLE (and only if no latched error). *)
        IF fbTrigStart.Q AND NOT stAuto.bError THEN
            stAuto.eStep := E_AutoStep.EXTENDING;
        END_IF

    E_AutoStep.EXTENDING:
        bCmdExtend  := TRUE;
        bCmdRetract := FALSE;
        stHmi.eMode := E_ControlMode.Automatic;
        IF stCfg.bNoSensors THEN
            (* Sensorless: PT = extend duration; timer expiry = success. *)
            IF fbTimerExtend.Q THEN
                stAuto.eStep := E_AutoStep.DWELL_EXT;
            END_IF
        ELSE
            (* Feedback mismatch = physical impossibility, sensor fault. *)
            IF stHmi.bIsExtended AND stHmi.bIsRetracted THEN
                stAuto.bError     := TRUE;
                stAuto.sErrorText := 'Both sensors active during EXTENDING (feedback mismatch)';
                stAuto.eStep      := E_AutoStep.ERR;
            ELSIF stHmi.bIsExtended THEN
                stAuto.eStep := E_AutoStep.DWELL_EXT;
            ELSIF fbTimerExtend.Q THEN
                stAuto.bError     := TRUE;
                stAuto.sErrorText := 'Timeout waiting for extended sensor';
                stAuto.eStep      := E_AutoStep.ERR;
            END_IF
        END_IF

    E_AutoStep.DWELL_EXT:
        (* Coil released — piston sits at the extended end sensor. *)
        bCmdExtend  := FALSE;
        bCmdRetract := FALSE;
        stHmi.eMode := E_ControlMode.Automatic;
        IF fbTimerDwellE.Q THEN
            stAuto.eStep := E_AutoStep.RETRACTING;
        END_IF

    E_AutoStep.RETRACTING:
        bCmdExtend  := FALSE;
        bCmdRetract := TRUE;
        stHmi.eMode := E_ControlMode.Automatic;
        IF stCfg.bNoSensors THEN
            (* Sensorless: PT = retract duration; timer expiry = success. *)
            IF fbTimerRetract.Q THEN
                stAuto.eStep := E_AutoStep.DWELL_RET;
            END_IF
        ELSE
            IF stHmi.bIsExtended AND stHmi.bIsRetracted THEN
                stAuto.bError     := TRUE;
                stAuto.sErrorText := 'Both sensors active during RETRACTING (feedback mismatch)';
                stAuto.eStep      := E_AutoStep.ERR;
            ELSIF stHmi.bIsRetracted THEN
                stAuto.eStep := E_AutoStep.DWELL_RET;
            ELSIF fbTimerRetract.Q THEN
                stAuto.bError     := TRUE;
                stAuto.sErrorText := 'Timeout waiting for retracted sensor';
                stAuto.eStep      := E_AutoStep.ERR;
            END_IF
        END_IF

    E_AutoStep.DWELL_RET:
        bCmdExtend  := FALSE;
        bCmdRetract := FALSE;
        stHmi.eMode := E_ControlMode.Automatic;
        IF fbTimerDwellR.Q THEN
            (* One complete cycle just ended. Count it. *)
            stAuto.nCyclesCompleted := stAuto.nCyclesCompleted + 1;
            IF stCfg.bContinuous THEN
                stAuto.eStep := E_AutoStep.EXTENDING;
            ELSE
                stAuto.eStep := E_AutoStep.IDLE;
            END_IF
        END_IF

    E_AutoStep.ERR:
        (* Latched error — outputs safe, wait for Ack or Reset. *)
        bCmdExtend  := FALSE;
        bCmdRetract := FALSE;
        (* Do NOT touch stHmi.eMode — let the operator flip to Manual for recovery. *)

END_CASE

(* ==========================================
   4. STEP-CHANGE DETECTION, LOGGING & ELAPSED TIMER
   Placed AFTER the state machine so we detect this cycle's transitions.
   fbStepTimer.IN := NOT bStepChanged pulses its ET back to 0 for one cycle
   on transition, then counts up until the next transition.
   ========================================== *)
bStepChanged := (stAuto.eStep <> ePrevStep);

(* Log every transition. ERR entries carry the human-readable sErrorText;
   all other transitions produce "PREV -> NEW" (relies on E_AutoStep's
   'to_string' attribute for label lookup). Runs AFTER bStepChanged is set
   but BEFORE ePrevStep is overwritten so we still have both endpoints. *)
IF bStepChanged THEN
    IF stAuto.eStep = E_AutoStep.ERR THEN
        F_LogEvent(eSev := E_LogSev.ERR, sSource := sName, sMsg := stAuto.sErrorText);
    ELSE
        F_LogEvent(
            eSev    := E_LogSev.INFO,
            sSource := sName,
            sMsg    := CONCAT(CONCAT(TO_STRING(ePrevStep), ' -> '), TO_STRING(stAuto.eStep))
        );
    END_IF
END_IF

ePrevStep := stAuto.eStep;

fbStepTimer(IN := NOT bStepChanged, PT := T#1D);
stAuto.tElapsedS := DINT_TO_LREAL(TIME_TO_DINT(fbStepTimer.ET)) * 0.001;

(* ==========================================
   5. STATUS TEXT MIRROR — refresh sStepText every cycle
   ========================================== *)
CASE stAuto.eStep OF
    E_AutoStep.IDLE:       stAuto.sStepText := 'Idle';
    E_AutoStep.EXTENDING:  stAuto.sStepText := 'Extending';
    E_AutoStep.DWELL_EXT:  stAuto.sStepText := 'Dwell (extended)';
    E_AutoStep.RETRACTING: stAuto.sStepText := 'Retracting';
    E_AutoStep.DWELL_RET:  stAuto.sStepText := 'Dwell (retracted)';
    E_AutoStep.ERR:        stAuto.sStepText := 'ERROR';
ELSE
    stAuto.sStepText := 'Unknown';
END_CASE

END_FUNCTION_BLOCK

// ---- POUs/F_LogEvent.TcPOU
(*
    Push one entry into the GVL_Log ring buffer.

    Callable from any scan without side effects on control logic. DEBUG entries
    are dropped when GVL_Log.bDebugMode = FALSE, so leaving DBG calls in
    production code costs nothing.

    Returns TRUE if the entry was recorded, FALSE if dropped by the debug filter.
*)
FUNCTION F_LogEvent : BOOL
VAR_INPUT
    eSev    : E_LogSev;
    sSource : STRING(20);
    sMsg    : STRING(80);
END_VAR
VAR
    idx : UDINT;
    k   : INT;
END_VAR

// Global mute — operator can disable ALL PLC logging from the HMI. When
// FALSE, we drop the event silently; the ring buffer and aRecent mirror
// are not touched so the last-known state stays visible.
IF NOT GVL_Log.bLogEnabled THEN
    F_LogEvent := FALSE;
    RETURN;
END_IF

// Debug filter — drop DBG severity when debug mode is off
IF (eSev = E_LogSev.DBG) AND NOT GVL_Log.bDebugMode THEN
    F_LogEvent := FALSE;
    RETURN;
END_IF

// Write into the ring at slot = nWriteIdx MOD 256
idx := GVL_Log.nWriteIdx MOD 256;
GVL_Log.aLog[idx].eSev    := eSev;
GVL_Log.aLog[idx].sSource := sSource;
GVL_Log.aLog[idx].sMsg    := sMsg;

// Shift the newest-first mirror down by one and write the new entry at
// [0]. HMI Logs page binds aRecent[0..19] directly in display order.
FOR k := 19 TO 1 BY -1 DO
    GVL_Log.aRecent[k] := GVL_Log.aRecent[k-1];
END_FOR
GVL_Log.aRecent[0].eSev    := eSev;
GVL_Log.aRecent[0].sSource := sSource;
GVL_Log.aRecent[0].sMsg    := sMsg;

// Increment the monotonic write counter — Python bridge polls this and
// drains any slots between its lastReadIdx and this value.
GVL_Log.nWriteIdx := GVL_Log.nWriteIdx + 1;

F_LogEvent := TRUE;

END_FUNCTION

// ---- POUs/FB_MasterAutoCycle.TcPOU
FUNCTION_BLOCK FB_MasterAutoCycle
(* Full-machine coordinated auto sequence spanning the robot and the 3
   pairs of SepSol / PushSol pistons (pair count fixed at 3 for this
   machine).

   Robot interface (TCP-only, 2026-07-26). The former discrete-I/O handshake
   is retired. All robot-side signals travel over FB_RobotTcpClient's
   STATE:n / CMD:n protocol:

     Robot -> PLC   nRobotCmd in {1,2}  (1=start, 2=reset error)
                    MAIN R_TRIGs on the edges; start pulse arrives here as
                    the VAR_INPUT bExtStartPulse.
     PLC -> Robot   nStateOut = TO_INT(eStep) or MANUAL(30)
                    Written by MAIN each scan, pushed by FB_RobotTcpClient
                    on change and as keep-alive.

   The cycle starts on any rising edge of bExtStartPulse (robot cmd=1, one
   scan wide), the HMI START button, or the sim-start flag.

   Sequence (all 3 Sep/Push pairs move in parallel; both grips move together):

     IDLE                    START button OR bExtStartPulse pulse OR SimIdle
                             OR bContinuous checked (level - keeps re-arming)
     INIT_PUSH_RETRACTING    drive PushCmdRetract[1..3]; wait AND of all
                             PushIsRetracted. Guarantees pistons are home before
                             a cycle starts, even if a prior manual move left
                             them extended.
     INIT_SEP_RETRACTING     drive SepCmdRetract[1..3]; wait AND of all
                             SepIsRetracted. Push must retract first (see INIT
                             above) because sep retract with push extended is
                             the same collision case avoided end-of-cycle.
     INIT_GRIP_RETRACTING    drive GripCmdRetract[1..2]; wait AND of all
                             GripIsRetracted. Defensive symmetry with the INIT
                             Sep/Push states, so a manual jog left extended
                             does not collide with the arriving plate.
     WAIT_PLATE              wait bPlateSenL AND bPlateSenR (robot has placed
                             the plate on the fixture). Latched at start only;
                             sensors are not monitored past this step.
     GRIP_EXTENDING          drive GripCmdExtend[1..2]; wait AND of all
                             GripIsExtended. Plate is clamped from both sides.
     SEP_EXTENDING           drive SepCmdExtend[1..3]; wait AND of all SepIsExtended.
                             Grip stays extended for every state below.
     PUSH_EXTENDING          drive PushCmdExtend[1..3]; wait AND of all PushIsExtended
     DWELL_PUSH              hold both extended; wait tDwellPushMs
     PUSH_RETRACTING         drive PushCmdRetract[1..3]; wait AND of all PushIsRetracted
     PUSH_RETRACTED_DWELL    wait tPushRetractedDwellMs
     SEP_RETRACTING          drive SepCmdRetract[1..3]; wait AND of all SepIsRetracted
     SEP_RETRACTED_DWELL     wait tSepRetractedDwellMs
     GRIP_RETRACTING         drive GripCmdRetract[1..2]; wait AND of all
                             GripIsRetracted. Releases the plate; increment
                             nCyclesCompleted; back to IDLE.
     ERR                     latched; iErrorCode set to step code; bContinuous
                             cleared so RESET does not restart motion.
                             Reset on HMI RESET rising edge.

   Error codes:
     0  = OK
     1  = SEP_EXTENDING timed out
     3  = PUSH_EXTENDING timed out
     4  = PUSH_RETRACTING timed out
     5  = SEP_RETRACTING timed out
     6  = INIT_PUSH_RETRACTING timed out
     7  = INIT_SEP_RETRACTING timed out
     8  = INIT_GRIP_RETRACTING timed out
     9  = WAIT_PLATE timed out (plate never arrived / one sensor never TRUE)
    10  = GRIP_EXTENDING timed out
    11  = GRIP_RETRACTING timed out
    99  = Operator STOP while running

   The former WAIT_POS2 state (error code 2) is retired: the robot code
   (src0.lua PerformStandSequence) already moves the arm clear of the
   stand BEFORE raising STAND_SEQ_DO, so the PLC does not need a separate
   "robot moved away" wait between SEP_EXTENDING and PUSH_EXTENDING. The
   E_MasterAutoStep.WAIT_POS2 enum value and stHmi.bSimStep_WaitPos2 flag
   remain declared but are unused; safe to remove once the HMI is cleaned.

   Per-step Sim flags on stHmi (bSimStep_Idle, bSimStep_SepExt, and so on)
   let a bench operator advance any waiting step without physical sensors.
   Rising-edge triggered; the FB auto-clears the flag after consumption.

   Sensorless mode (stCfg.bNoSensors): the 4 movement states ignore sensor
   feedback and advance when tStepTimeoutMs expires — the timeout doubles
   as the fixed step duration. Error codes 1/3/4/5 cannot occur while
   sensorless. *)
VAR_INPUT
    (* External start pulse (rising-edge; one scan wide). MAIN fires this
       when the robot's CMD:1 arrives via TCP, or a physical PB1 rising
       edge in Auto mode. HMI START button and SimStartAssembly are
       consumed separately below via their own R_TRIGs. *)
    bExtStartPulse        : BOOL;

    (* Global machine-mode gate (stCfg.bAutoMode). While FALSE the cycle is
       held in IDLE: every start trigger is ignored and a running cycle is
       aborted back to IDLE. This is the hard interlock that stops the
       operator or a stray robot edge starting motion while the machine is
       in Manual. *)
    bMachineAuto          : BOOL;

    (* Per-pair sensor state. MAIN wires each element from stSepSolK/stPushSolK.bIs*. *)
    bSepIsExtended        : ARRAY[1..3] OF BOOL;
    bSepIsRetracted       : ARRAY[1..3] OF BOOL;
    bPushIsExtended       : ARRAY[1..3] OF BOOL;
    bPushIsRetracted      : ARRAY[1..3] OF BOOL;

    (* Grip pistons — L=[1], R=[2]. MAIN wires from stGripSolL/R.bIs*. *)
    bGripIsExtended       : ARRAY[1..2] OF BOOL;
    bGripIsRetracted      : ARRAY[1..2] OF BOOL;

    (* Plate-presence sensors gating WAIT_PLATE. Both must be TRUE before the
       cycle can advance out of WAIT_PLATE into GRIP_EXTENDING. Latched at
       cycle start only — not monitored past that step. *)
    bPlateSenL            : BOOL;
    bPlateSenR            : BOOL;
END_VAR

VAR_IN_OUT
    stHmi     : ST_HmiMasterAuto;
    stCfg     : ST_HmiMasterAutoCfg;
    stRobot   : ST_HmiRobot;
END_VAR

VAR_OUTPUT
    (* MAIN OR-merges these with the per-piston auto FBs. *)
    bSepCmdExtend         : ARRAY[1..3] OF BOOL;
    bSepCmdRetract        : ARRAY[1..3] OF BOOL;
    bPushCmdExtend        : ARRAY[1..3] OF BOOL;
    bPushCmdRetract       : ARRAY[1..3] OF BOOL;

    (* Grip piston commands. Extend held TRUE from GRIP_EXTENDING through
       SEP_RETRACTED_DWELL so the plate stays clamped for the entire cycle. *)
    bGripCmdExtend        : ARRAY[1..2] OF BOOL;
    bGripCmdRetract       : ARRAY[1..2] OF BOOL;

    (* TRUE while the master cycle is in any state other than IDLE or ERR.
       MAIN reads this to force enabled pistons' stHmi.eMode := Automatic
       while running, so bAutoCmd* actually reaches the piston coil (in
       Manual mode the piston FB ignores bAutoCmd*)
    bAnyRunning           : BOOL;
END_VAR

VAR
    (* Rising-edge detectors for momentary HMI buttons + robot start signal. *)
    fbTrigStart           : R_TRIG;
    fbTrigStop            : R_TRIG;
    fbTrigReset           : R_TRIG;
    fbTrigStartAssembly   : R_TRIG;

    (* Rising-edge detectors for per-step Sim flags. *)
    fbSim_Idle            : R_TRIG;
    fbSim_InitPushRet     : R_TRIG;
    fbSim_InitSepRet      : R_TRIG;
    fbSim_InitGripRet     : R_TRIG;
    fbSim_WaitPlate       : R_TRIG;
    fbSim_GripExt         : R_TRIG;
    fbSim_SepExt          : R_TRIG;
    fbSim_PushExt         : R_TRIG;
    fbSim_DwellPush       : R_TRIG;
    fbSim_PushRet         : R_TRIG;
    fbSim_PushRetDwell    : R_TRIG;
    fbSim_SepRet          : R_TRIG;
    fbSim_SepRetDwell     : R_TRIG;
    fbSim_GripRet         : R_TRIG;

    (* Per-step timer. Same TON, different PT depending on state. On DWELL
       states PT is the dwell; on wait states PT is the timeout. *)
    tonStep               : TON;
    ePrevStep             : E_MasterAutoStep;   (* transition detect for timer reset *)

    (* Loop index *)
    i                     : USINT;

    (* Aggregate sensor flags, computed each cycle in Section 1. *)
    bAllSepExtended       : BOOL;
    bAllSepRetracted      : BOOL;
    bAllPushExtended      : BOOL;
    bAllPushRetracted     : BOOL;
    bAllGripExtended      : BOOL;
    bAllGripRetracted     : BOOL;
    bPlateOk              : BOOL;
END_VAR

(* ==========================================
   0a. RISING-EDGE DETECTORS
   ========================================== *)
fbTrigStart        (CLK := stHmi.bStart);
fbTrigStop         (CLK := stHmi.bStop);
fbTrigReset        (CLK := stHmi.bReset);
fbTrigStartAssembly(CLK := stHmi.bSimStartAssembly);

fbSim_Idle        (CLK := stHmi.bSimStep_Idle);
fbSim_InitPushRet (CLK := stHmi.bSimStep_InitPushRet);
fbSim_InitSepRet  (CLK := stHmi.bSimStep_InitSepRet);
fbSim_InitGripRet (CLK := stHmi.bSimStep_InitGripRet);
fbSim_WaitPlate   (CLK := stHmi.bSimStep_WaitPlate);
fbSim_GripExt     (CLK := stHmi.bSimStep_GripExt);
fbSim_SepExt      (CLK := stHmi.bSimStep_SepExt);
fbSim_PushExt     (CLK := stHmi.bSimStep_PushExt);
fbSim_DwellPush   (CLK := stHmi.bSimStep_DwellPush);
fbSim_PushRet     (CLK := stHmi.bSimStep_PushRet);
fbSim_PushRetDwell(CLK := stHmi.bSimStep_PushRetDwell);
fbSim_SepRet      (CLK := stHmi.bSimStep_SepRet);
fbSim_SepRetDwell (CLK := stHmi.bSimStep_SepRetDwell);
fbSim_GripRet     (CLK := stHmi.bSimStep_GripRet);

(* ==========================================
   0b. AUTO-CLEAR ONE-SHOT FLAGS ON RISING EDGE
   HMI button flags and Sim flags are momentary; after we detect the
   rising edge we clear the raw flag so the operator's next click can
   fire again. bExtStartPulse is already a one-scan pulse produced by
   MAIN's R_TRIG on the robot's TCP command channel -- nothing to clear.
   ========================================== *)
IF fbTrigStart.Q  THEN
    stHmi.bStart := FALSE;
    F_LogEvent(eSev := E_LogSev.INFO, sSource := stHmi.Name, sMsg := 'START pressed');
END_IF;
IF fbTrigStop.Q   THEN
    stHmi.bStop  := FALSE;
    F_LogEvent(eSev := E_LogSev.INFO, sSource := stHmi.Name, sMsg := 'STOP pressed');
END_IF;
IF fbTrigReset.Q  THEN
    stHmi.bReset := FALSE;
    F_LogEvent(eSev := E_LogSev.INFO, sSource := stHmi.Name, sMsg := 'RESET pressed');
END_IF;

(* Bench sim of the robot start: fires on the HMI checkbox rising edge and
   auto-clears. Log so bench-driven cycles show up in the event log. The
   robot-driven start comes in as bExtStartPulse (already an edge, no R_TRIG
   needed here) and is logged from MAIN when nRobotCmd goes 0->1. *)
IF fbTrigStartAssembly.Q THEN
    stHmi.bSimStartAssembly := FALSE;
    F_LogEvent(eSev := E_LogSev.INFO, sSource := stHmi.Name, sMsg := 'Sim start pressed');
END_IF;
IF bExtStartPulse THEN
    F_LogEvent(eSev := E_LogSev.INFO, sSource := stHmi.Name, sMsg := 'External start pulse');
END_IF;

IF fbSim_Idle.Q         THEN stHmi.bSimStep_Idle         := FALSE; END_IF;
IF fbSim_InitPushRet.Q  THEN stHmi.bSimStep_InitPushRet  := FALSE; END_IF;
IF fbSim_InitSepRet.Q   THEN stHmi.bSimStep_InitSepRet   := FALSE; END_IF;
IF fbSim_InitGripRet.Q  THEN stHmi.bSimStep_InitGripRet  := FALSE; END_IF;
IF fbSim_WaitPlate.Q    THEN stHmi.bSimStep_WaitPlate    := FALSE; END_IF;
IF fbSim_GripExt.Q      THEN stHmi.bSimStep_GripExt      := FALSE; END_IF;
IF fbSim_SepExt.Q       THEN stHmi.bSimStep_SepExt       := FALSE; END_IF;
IF fbSim_PushExt.Q      THEN stHmi.bSimStep_PushExt      := FALSE; END_IF;
IF fbSim_DwellPush.Q    THEN stHmi.bSimStep_DwellPush    := FALSE; END_IF;
IF fbSim_PushRet.Q      THEN stHmi.bSimStep_PushRet      := FALSE; END_IF;
IF fbSim_PushRetDwell.Q THEN stHmi.bSimStep_PushRetDwell := FALSE; END_IF;
IF fbSim_SepRet.Q       THEN stHmi.bSimStep_SepRet       := FALSE; END_IF;
IF fbSim_SepRetDwell.Q  THEN stHmi.bSimStep_SepRetDwell  := FALSE; END_IF;
IF fbSim_GripRet.Q      THEN stHmi.bSimStep_GripRet      := FALSE; END_IF;

(* ==========================================
   1. AGGREGATE SENSOR STATE
   ========================================== *)
bAllSepExtended   := bSepIsExtended[1]   AND bSepIsExtended[2]   AND bSepIsExtended[3];
bAllSepRetracted  := bSepIsRetracted[1]  AND bSepIsRetracted[2]  AND bSepIsRetracted[3];
bAllPushExtended  := bPushIsExtended[1]  AND bPushIsExtended[2]  AND bPushIsExtended[3];
bAllPushRetracted := bPushIsRetracted[1] AND bPushIsRetracted[2] AND bPushIsRetracted[3];
bAllGripExtended  := bGripIsExtended[1]  AND bGripIsExtended[2];
bAllGripRetracted := bGripIsRetracted[1] AND bGripIsRetracted[2];
bPlateOk          := bPlateSenL AND bPlateSenR;

(* ==========================================
   2. GLOBAL OVERRIDES — STOP and RESET
   STOP while running latches error 99 and drops to ERR. HMI RESET clears
   the error and returns to IDLE. The robot's own RESET_ALARM (robot DI 10)
   is handled robot-side; the PLC does not receive it in the discrete-IO
   interface. Operator must reset both sides after a fault.
   ========================================== *)
IF fbTrigStop.Q AND stHmi.eStep <> E_MasterAutoStep.IDLE AND stHmi.eStep <> E_MasterAutoStep.ERR THEN
    stHmi.iErrorCode := 99;
    stHmi.sErrorText := 'Operator STOP while running';
    stHmi.eStep      := E_MasterAutoStep.ERR;
    (* Drop Continuous on any ERR entry so RESET does not instantly
       restart motion with the box still checked. *)
    stCfg.bContinuous := FALSE;
END_IF;

IF fbTrigReset.Q AND stHmi.eStep = E_MasterAutoStep.ERR THEN
    stHmi.iErrorCode := 0;
    stHmi.sErrorText := '';
    stHmi.eStep      := E_MasterAutoStep.IDLE;
END_IF;

(* Global Auto/Manual hard interlock. Switching the machine to Manual (or
   being in Manual) forces the cycle back to IDLE from any running state and
   drops Continuous, so a stray robot start pulse cannot restart motion.
   Not treated as a fault (no ERR/error code) — Manual is a normal operator
   choice, not an alarm. ERR stays latched until RESET. *)
IF NOT bMachineAuto AND stHmi.eStep <> E_MasterAutoStep.IDLE AND stHmi.eStep <> E_MasterAutoStep.ERR THEN
    stCfg.bContinuous := FALSE;
    stHmi.eStep       := E_MasterAutoStep.IDLE;
END_IF;

(* ==========================================
   3. STEP TIMER + TRANSITION LOG
   Reset tonStep on any state change. In DWELL states PT is the dwell
   duration and Q rising = "dwell complete, advance". In wait states PT
   is the timeout and Q rising = "timed out, error". Non-waiting states
   (IDLE, ERR) do not consult Q.

   Also emit one log entry per transition — INFO with "PREV -> NEW" for
   normal advances, ERR with sErrorText when the new state is ERR. The
   check runs one scan AFTER Section 4 set eStep, so sErrorText and
   iErrorCode are already populated. Order matters: log BEFORE updating
   ePrevStep so both endpoints are still available.
   ========================================== *)
IF stHmi.eStep <> ePrevStep THEN
    IF stHmi.eStep = E_MasterAutoStep.ERR THEN
        F_LogEvent(eSev := E_LogSev.ERR, sSource := stHmi.Name, sMsg := stHmi.sErrorText);
    ELSE
        F_LogEvent(
            eSev    := E_LogSev.INFO,
            sSource := stHmi.Name,
            sMsg    := CONCAT(CONCAT(TO_STRING(ePrevStep), ' -> '), TO_STRING(stHmi.eStep))
        );
    END_IF

    tonStep(IN := FALSE, PT := T#0MS);   // pulse-off resets ET to 0
    ePrevStep := stHmi.eStep;
END_IF;

(* PT depends on state. Wait states use tStepTimeoutMs; dwell states use their own.
   WAIT_PLATE uses tPlateWaitTimeoutMs (bounded by robot placement time). *)
CASE stHmi.eStep OF
    E_MasterAutoStep.DWELL_PUSH:
        tonStep(IN := TRUE, PT := UDINT_TO_TIME(stCfg.tDwellPushMs));
    E_MasterAutoStep.PUSH_RETRACTED_DWELL:
        tonStep(IN := TRUE, PT := UDINT_TO_TIME(stCfg.tPushRetractedDwellMs));
    E_MasterAutoStep.SEP_RETRACTED_DWELL:
        tonStep(IN := TRUE, PT := UDINT_TO_TIME(stCfg.tSepRetractedDwellMs));
    E_MasterAutoStep.WAIT_PLATE:
        tonStep(IN := TRUE, PT := UDINT_TO_TIME(stCfg.tPlateWaitTimeoutMs));
    E_MasterAutoStep.SEP_EXTENDING,
    E_MasterAutoStep.PUSH_EXTENDING,
    E_MasterAutoStep.PUSH_RETRACTING,
    E_MasterAutoStep.SEP_RETRACTING,
    E_MasterAutoStep.INIT_PUSH_RETRACTING,
    E_MasterAutoStep.INIT_SEP_RETRACTING,
    E_MasterAutoStep.INIT_GRIP_RETRACTING,
    E_MasterAutoStep.GRIP_EXTENDING,
    E_MasterAutoStep.GRIP_RETRACTING:
        tonStep(IN := TRUE, PT := UDINT_TO_TIME(stCfg.tStepTimeoutMs));
ELSE
    tonStep(IN := FALSE, PT := T#0MS);
END_CASE;

stHmi.tElapsedS := DINT_TO_LREAL(TIME_TO_DINT(tonStep.ET)) / 1000.0;

(* ==========================================
   4. STATE MACHINE
   Default: clear all commands each cycle in the ELSE-ish paths so a
   dropped state doesn't leave stale coils driven. Each state re-asserts
   the commands it owns. Grip commands are held TRUE from GRIP_EXTENDING
   through SEP_RETRACTED_DWELL so the plate stays clamped for the entire
   Sep/Push cycle.
   ========================================== *)
CASE stHmi.eStep OF

    E_MasterAutoStep.IDLE:
        FOR i := 1 TO 3 DO
            bSepCmdExtend[i]   := FALSE;
            bSepCmdRetract[i]  := FALSE;
            bPushCmdExtend[i]  := FALSE;
            bPushCmdRetract[i] := FALSE;
        END_FOR;
        FOR i := 1 TO 2 DO
            bGripCmdExtend[i]  := FALSE;
            bGripCmdRetract[i] := FALSE;
        END_FOR;
        (* No active error while in IDLE (unless just about to enter ERR
           via a global override, handled above). *)
        stHmi.iErrorCode := 0;
        stHmi.sErrorText := '';

        IF bMachineAuto AND (fbTrigStart.Q OR bExtStartPulse OR fbTrigStartAssembly.Q OR fbSim_Idle.Q OR stCfg.bContinuous) THEN
            (* Robot (via TCP CMD:1 -> MAIN R_TRIG -> bExtStartPulse),
               operator (fbTrigStart), or bench sim (fbTrigStartAssembly)
               has requested a cycle. Gated by bMachineAuto: in Manual the
               machine cannot start, even on a robot start pulse (no
               double-control). While bContinuous is checked, IDLE starts
               the next cycle immediately — no external edge needed.

               Enter INIT_PUSH_RETRACTING first (not SEP_EXTENDING directly)
               so pistons left extended by a prior manual move are driven
               home before the cycle proper starts. If everything is already
               retracted, the three INIT states self-satisfy on the next scan. *)
            stHmi.eStep := E_MasterAutoStep.INIT_PUSH_RETRACTING;
        END_IF;

    E_MasterAutoStep.INIT_PUSH_RETRACTING:
        (* Mirror end-of-cycle PUSH_RETRACTING: assert push retract only. Sep
           stays uncommanded (whatever position it was left in — its retract
           follows in INIT_SEP_RETRACTING). Grip uncommanded here. *)
        FOR i := 1 TO 3 DO
            bSepCmdExtend[i]   := FALSE;
            bSepCmdRetract[i]  := FALSE;
            bPushCmdExtend[i]  := FALSE;
            bPushCmdRetract[i] := TRUE;
        END_FOR;
        FOR i := 1 TO 2 DO
            bGripCmdExtend[i]  := FALSE;
            bGripCmdRetract[i] := FALSE;
        END_FOR;

        IF bAllPushRetracted OR fbSim_InitPushRet.Q OR (stCfg.bNoSensors AND tonStep.Q) THEN
            stHmi.eStep := E_MasterAutoStep.INIT_SEP_RETRACTING;
        ELSIF tonStep.Q THEN
            stHmi.iErrorCode := 6;
            stHmi.sErrorText := 'INIT_PUSH_RETRACTING timed out';
            stHmi.eStep := E_MasterAutoStep.ERR;
            stCfg.bContinuous := FALSE;
        END_IF;

    E_MasterAutoStep.INIT_SEP_RETRACTING:
        (* Push is confirmed home; now retract sep. *)
        FOR i := 1 TO 3 DO
            bSepCmdExtend[i]   := FALSE;
            bSepCmdRetract[i]  := TRUE;
            bPushCmdExtend[i]  := FALSE;
            bPushCmdRetract[i] := FALSE;
        END_FOR;
        FOR i := 1 TO 2 DO
            bGripCmdExtend[i]  := FALSE;
            bGripCmdRetract[i] := FALSE;
        END_FOR;

        IF bAllSepRetracted OR fbSim_InitSepRet.Q OR (stCfg.bNoSensors AND tonStep.Q) THEN
            stHmi.eStep := E_MasterAutoStep.INIT_GRIP_RETRACTING;
        ELSIF tonStep.Q THEN
            stHmi.iErrorCode := 7;
            stHmi.sErrorText := 'INIT_SEP_RETRACTING timed out';
            stHmi.eStep := E_MasterAutoStep.ERR;
            stCfg.bContinuous := FALSE;
        END_IF;

    E_MasterAutoStep.INIT_GRIP_RETRACTING:
        (* Both Sep and Push confirmed home; now retract grip. Defensive
           symmetry with INIT_PUSH_RETRACTING / INIT_SEP_RETRACTING so a
           prior manual jog does not leave grip clamped when the plate
           arrives. *)
        FOR i := 1 TO 3 DO
            bSepCmdExtend[i]   := FALSE;
            bSepCmdRetract[i]  := FALSE;
            bPushCmdExtend[i]  := FALSE;
            bPushCmdRetract[i] := FALSE;
        END_FOR;
        FOR i := 1 TO 2 DO
            bGripCmdExtend[i]  := FALSE;
            bGripCmdRetract[i] := TRUE;
        END_FOR;

        IF bAllGripRetracted OR fbSim_InitGripRet.Q OR (stCfg.bNoSensors AND tonStep.Q) THEN
            stHmi.eStep := E_MasterAutoStep.WAIT_PLATE;
        ELSIF tonStep.Q THEN
            stHmi.iErrorCode := 8;
            stHmi.sErrorText := 'INIT_GRIP_RETRACTING timed out';
            stHmi.eStep := E_MasterAutoStep.ERR;
            stCfg.bContinuous := FALSE;
        END_IF;

    E_MasterAutoStep.WAIT_PLATE:
        (* Nothing driven — waiting for the robot to place the plate on the
           fixture. Both plate sensors must confirm TRUE before advancing.
           No sensorless fallback: the whole point of this state is to gate
           on the plate presence. Timeout uses tPlateWaitTimeoutMs (see
           Section 3 timer selector). *)
        FOR i := 1 TO 3 DO
            bSepCmdExtend[i]   := FALSE;
            bSepCmdRetract[i]  := FALSE;
            bPushCmdExtend[i]  := FALSE;
            bPushCmdRetract[i] := FALSE;
        END_FOR;
        FOR i := 1 TO 2 DO
            bGripCmdExtend[i]  := FALSE;
            bGripCmdRetract[i] := FALSE;
        END_FOR;

        IF bPlateOk OR fbSim_WaitPlate.Q THEN
            stHmi.eStep := E_MasterAutoStep.GRIP_EXTENDING;
        ELSIF tonStep.Q THEN
            stHmi.iErrorCode := 9;
            stHmi.sErrorText := 'WAIT_PLATE timed out (plate never arrived)';
            stHmi.eStep := E_MasterAutoStep.ERR;
            stCfg.bContinuous := FALSE;
        END_IF;

    E_MasterAutoStep.GRIP_EXTENDING:
        (* Plate is on the fixture; clamp it from both sides. *)
        FOR i := 1 TO 2 DO
            bGripCmdExtend[i]  := TRUE;
            bGripCmdRetract[i] := FALSE;
        END_FOR;

        IF bAllGripExtended OR fbSim_GripExt.Q OR (stCfg.bNoSensors AND tonStep.Q) THEN
            stHmi.eStep := E_MasterAutoStep.SEP_EXTENDING;
        ELSIF tonStep.Q THEN
            stHmi.iErrorCode := 10;
            stHmi.sErrorText := 'GRIP_EXTENDING timed out';
            stHmi.eStep := E_MasterAutoStep.ERR;
            stCfg.bContinuous := FALSE;
        END_IF;

    E_MasterAutoStep.SEP_EXTENDING:
        FOR i := 1 TO 3 DO
            bSepCmdExtend[i]  := TRUE;
            bSepCmdRetract[i] := FALSE;
        END_FOR;
        FOR i := 1 TO 2 DO
            bGripCmdExtend[i] := TRUE;   (* hold grip clamped *)
        END_FOR;

        IF bAllSepExtended OR fbSim_SepExt.Q OR (stCfg.bNoSensors AND tonStep.Q) THEN
            (* Skip the former WAIT_POS2 — the robot has already moved clear
               of the stand before signaling start via TCP CMD:1. *)
            stHmi.eStep := E_MasterAutoStep.PUSH_EXTENDING;
        ELSIF tonStep.Q THEN   (* only reachable when NOT bNoSensors *)
            stHmi.iErrorCode := 1;
            stHmi.sErrorText := 'SEP_EXTENDING timed out';
            stHmi.eStep := E_MasterAutoStep.ERR;
            stCfg.bContinuous := FALSE;
        END_IF;

    E_MasterAutoStep.PUSH_EXTENDING:
        FOR i := 1 TO 3 DO
            bSepCmdExtend[i]   := TRUE;   (* hold sep out *)
            bPushCmdExtend[i]  := TRUE;
            bPushCmdRetract[i] := FALSE;
        END_FOR;
        FOR i := 1 TO 2 DO
            bGripCmdExtend[i] := TRUE;
        END_FOR;

        IF bAllPushExtended OR fbSim_PushExt.Q OR (stCfg.bNoSensors AND tonStep.Q) THEN
            stHmi.eStep := E_MasterAutoStep.DWELL_PUSH;
        ELSIF tonStep.Q THEN
            stHmi.iErrorCode := 3;
            stHmi.sErrorText := 'PUSH_EXTENDING timed out';
            stHmi.eStep := E_MasterAutoStep.ERR;
            stCfg.bContinuous := FALSE;
        END_IF;

    E_MasterAutoStep.DWELL_PUSH:
        (* Hold everything out. *)
        FOR i := 1 TO 3 DO
            bSepCmdExtend[i]  := TRUE;
            bPushCmdExtend[i] := TRUE;
        END_FOR;
        FOR i := 1 TO 2 DO
            bGripCmdExtend[i] := TRUE;
        END_FOR;

        IF tonStep.Q OR fbSim_DwellPush.Q THEN
            stHmi.eStep := E_MasterAutoStep.PUSH_RETRACTING;
        END_IF;

    E_MasterAutoStep.PUSH_RETRACTING:
        (* Sep still extended, push retract command asserted. *)
        FOR i := 1 TO 3 DO
            bSepCmdExtend[i]   := TRUE;
            bPushCmdExtend[i]  := FALSE;
            bPushCmdRetract[i] := TRUE;
        END_FOR;
        FOR i := 1 TO 2 DO
            bGripCmdExtend[i] := TRUE;
        END_FOR;

        IF bAllPushRetracted OR fbSim_PushRet.Q OR (stCfg.bNoSensors AND tonStep.Q) THEN
            stHmi.eStep := E_MasterAutoStep.PUSH_RETRACTED_DWELL;
        ELSIF tonStep.Q THEN
            stHmi.iErrorCode := 4;
            stHmi.sErrorText := 'PUSH_RETRACTING timed out';
            stHmi.eStep := E_MasterAutoStep.ERR;
            stCfg.bContinuous := FALSE;
        END_IF;

    E_MasterAutoStep.PUSH_RETRACTED_DWELL:
        (* Sep still held extended, push commands cleared. *)
        FOR i := 1 TO 3 DO
            bSepCmdExtend[i]   := TRUE;
            bPushCmdExtend[i]  := FALSE;
            bPushCmdRetract[i] := FALSE;
        END_FOR;
        FOR i := 1 TO 2 DO
            bGripCmdExtend[i] := TRUE;
        END_FOR;

        IF tonStep.Q OR fbSim_PushRetDwell.Q THEN
            stHmi.eStep := E_MasterAutoStep.SEP_RETRACTING;
        END_IF;

    E_MasterAutoStep.SEP_RETRACTING:
        FOR i := 1 TO 3 DO
            bSepCmdExtend[i]  := FALSE;
            bSepCmdRetract[i] := TRUE;
        END_FOR;
        FOR i := 1 TO 2 DO
            bGripCmdExtend[i] := TRUE;
        END_FOR;

        IF bAllSepRetracted OR fbSim_SepRet.Q OR (stCfg.bNoSensors AND tonStep.Q) THEN
            stHmi.eStep := E_MasterAutoStep.SEP_RETRACTED_DWELL;
        ELSIF tonStep.Q THEN
            stHmi.iErrorCode := 5;
            stHmi.sErrorText := 'SEP_RETRACTING timed out';
            stHmi.eStep := E_MasterAutoStep.ERR;
            stCfg.bContinuous := FALSE;
        END_IF;

    E_MasterAutoStep.SEP_RETRACTED_DWELL:
        (* Sep/Push home; grip still clamped (released in GRIP_RETRACTING). *)
        FOR i := 1 TO 3 DO
            bSepCmdExtend[i]   := FALSE;
            bSepCmdRetract[i]  := FALSE;
            bPushCmdExtend[i]  := FALSE;
            bPushCmdRetract[i] := FALSE;
        END_FOR;
        FOR i := 1 TO 2 DO
            bGripCmdExtend[i] := TRUE;
        END_FOR;

        IF tonStep.Q OR fbSim_SepRetDwell.Q THEN
            stHmi.eStep := E_MasterAutoStep.GRIP_RETRACTING;
        END_IF;

    E_MasterAutoStep.GRIP_RETRACTING:
        (* Very last motion: release the plate. On successful retract,
           increment nCyclesCompleted and return to IDLE. *)
        FOR i := 1 TO 3 DO
            bSepCmdExtend[i]   := FALSE;
            bSepCmdRetract[i]  := FALSE;
            bPushCmdExtend[i]  := FALSE;
            bPushCmdRetract[i] := FALSE;
        END_FOR;
        FOR i := 1 TO 2 DO
            bGripCmdExtend[i]  := FALSE;
            bGripCmdRetract[i] := TRUE;
        END_FOR;

        IF bAllGripRetracted OR fbSim_GripRet.Q OR (stCfg.bNoSensors AND tonStep.Q) THEN
            stHmi.nCyclesCompleted := stHmi.nCyclesCompleted + 1;
            (* Back to IDLE. If bContinuous is still checked, IDLE re-arms
               the next cycle by itself on the next scan. *)
            stHmi.eStep := E_MasterAutoStep.IDLE;
        ELSIF tonStep.Q THEN
            stHmi.iErrorCode := 11;
            stHmi.sErrorText := 'GRIP_RETRACTING timed out';
            stHmi.eStep := E_MasterAutoStep.ERR;
            stCfg.bContinuous := FALSE;
        END_IF;

    E_MasterAutoStep.ERR:
        (* Latched. nStateOut mirrors ERR(99) so the robot's TCP client
           sees the fault via STATE:99 and can invoke its own error
           handler. Exit only via Section 2 (HMI RESET or CMD:2). *)
        FOR i := 1 TO 3 DO
            bSepCmdExtend[i]   := FALSE;
            bSepCmdRetract[i]  := FALSE;
            bPushCmdExtend[i]  := FALSE;
            bPushCmdRetract[i] := FALSE;
        END_FOR;
        FOR i := 1 TO 2 DO
            bGripCmdExtend[i]  := FALSE;
            bGripCmdRetract[i] := FALSE;
        END_FOR;

ELSE
    (* Defensive: any undefined value snaps to IDLE with no commands. *)
    FOR i := 1 TO 3 DO
        bSepCmdExtend[i]   := FALSE;
        bSepCmdRetract[i]  := FALSE;
        bPushCmdExtend[i]  := FALSE;
        bPushCmdRetract[i] := FALSE;
    END_FOR;
    FOR i := 1 TO 2 DO
        bGripCmdExtend[i]  := FALSE;
        bGripCmdRetract[i] := FALSE;
    END_FOR;
    stHmi.eStep := E_MasterAutoStep.IDLE;
END_CASE;

(* ==========================================
   5. STATUS MIRROR — human-readable step name + running flag
   TO_STRING relies on the enum's {to_string} attribute.
   bAnyRunning is TRUE any time the cycle is actively driving pistons —
   MAIN uses it to force enabled pistons into Automatic mode. False in ERR
   so the operator's manual choice is preserved after a fault.

   The "PLC is running" signal to the robot is derived robot-side from
   nStateOut != IDLE (see FB_RobotTcpClient); no separate outbound field
   needed here.
   ========================================== *)
stHmi.sStepText := TO_STRING(stHmi.eStep);
bAnyRunning     := (stHmi.eStep <> E_MasterAutoStep.IDLE)
               AND (stHmi.eStep <> E_MasterAutoStep.ERR);

END_FUNCTION_BLOCK

// ---- POUs/FB_SolSolPiston_2Pos.TcPOU
FUNCTION_BLOCK FB_SolSolPiston_2Pos
VAR_INPUT
    (* Automatic Commands from PLC sequence logic. Wired to FALSE in MAIN until FB_Auto exists. *)
    bAutoCmdExtend    : BOOL;
    bAutoCmdRetract   : BOOL;

    (* Physical Feedback (Proximity Switches) *)
    bSwitchExtended   : BOOL;
    bSwitchRetracted  : BOOL;
END_VAR

VAR_IN_OUT
    (* HMI contract — mode, manual + simulate inputs, latched + sensor status *)
    stHmi             : ST_HmiPiston;
END_VAR

VAR_OUTPUT
    (* Physical Outputs to Solenoids *)
    bOutSolenoidExtend  : BOOL;
    bOutSolenoidRetract : BOOL;
END_VAR

VAR
    (* Internal Target States *)
    bTargetExtend     : BOOL;
    bTargetRetract    : BOOL;

    (* HMI Manual-Button Edge Detection *)
    fbTrigManExtend   : R_TRIG;
    fbTrigManRetract  : R_TRIG;

    (* Effective sensor states = real OR HMI simulate. Recomputed every cycle in Section 0a. *)
    bSwitchExtended_eff  : BOOL;
    bSwitchRetracted_eff : BOOL;
END_VAR

(* ==========================================
   0a. EFFECTIVE SENSOR INPUTS (real OR HMI simulate)
   ========================================== *)
bSwitchExtended_eff  := bSwitchExtended  OR stHmi.bSimulateExtended;
bSwitchRetracted_eff := bSwitchRetracted OR stHmi.bSimulateRetracted;

(* ==========================================
   0. HMI MANUAL BUTTON LATCHING (Radio-Button Behavior)
   ========================================== *)
fbTrigManExtend(CLK := stHmi.bManCmdExtend);
fbTrigManRetract(CLK := stHmi.bManCmdRetract);

// Independent IFs (not ELSIF): if multiple edges fire in the same cycle, the last one wins (Retract > Extend).
IF fbTrigManExtend.Q  THEN stHmi.bSelectedExtend := TRUE;  stHmi.bSelectedRetract := FALSE; END_IF;
IF fbTrigManRetract.Q THEN stHmi.bSelectedExtend := FALSE; stHmi.bSelectedRetract := TRUE;  END_IF;

IF stHmi.eMode = E_ControlMode.Automatic THEN
    stHmi.bSelectedExtend := FALSE; stHmi.bSelectedRetract := FALSE;
END_IF;

(* ==========================================
   1. MODE SELECTION & COMMAND MAPPING
   ========================================== *)
IF stHmi.eMode = E_ControlMode.Automatic THEN
    bTargetExtend  := bAutoCmdExtend;
    bTargetRetract := bAutoCmdRetract;

ELSIF stHmi.eMode = E_ControlMode.Manual THEN
    bTargetExtend  := stHmi.bSelectedExtend;
    bTargetRetract := stHmi.bSelectedRetract;

ELSE
    // Safe default: undefined mode → no targets
    bTargetExtend  := FALSE;
    bTargetRetract := FALSE;
END_IF;

(* ==========================================
   1a. JOG OVERRIDE — clear latched selection while either jog is held
   ========================================== *)
// Section 1 above already copied stHmi.bSelected* into bTarget*. The stale
// bTarget* is harmless because Section 2's jog branches sit ahead of the
// bTarget* branches in the IF/ELSIF ladder and preempt them.
IF stHmi.bManJogExtend OR stHmi.bManJogRetract THEN
    stHmi.bSelectedExtend := FALSE; stHmi.bSelectedRetract := FALSE;
END_IF;

(* ==========================================
   1b. TARGET-REACHED RESET — clear bSelected* once the piston arrives
   ========================================== *)
IF stHmi.bSelectedExtend  AND bSwitchExtended_eff  THEN stHmi.bSelectedExtend  := FALSE; END_IF;
IF stHmi.bSelectedRetract AND bSwitchRetracted_eff THEN stHmi.bSelectedRetract := FALSE; END_IF;

(* ==========================================
   2. SOLENOID CONTROL — Jog takes priority over latched target
   ========================================== *)
// Jog branches first, gated by Manual mode. If both jogs are held
// simultaneously, Retract wins (matching the same-cycle collision rule
// in Section 0). Each branch still respects the corresponding effective
// sensor. In Automatic mode the jog branches are skipped entirely so
// bAutoCmd* controls the piston.

// JOG EXTEND: while held in Manual, drive Extend coil until end sensor
IF stHmi.bManJogExtend AND NOT bSwitchExtended_eff AND stHmi.eMode = E_ControlMode.Manual THEN
    bOutSolenoidExtend  := TRUE;
    bOutSolenoidRetract := FALSE;

// JOG RETRACT: while held in Manual, drive Retract coil until end sensor
ELSIF stHmi.bManJogRetract AND NOT bSwitchRetracted_eff AND stHmi.eMode = E_ControlMode.Manual THEN
    bOutSolenoidRetract := TRUE;
    bOutSolenoidExtend  := FALSE;

// CASE 1: Move to EXTENDED position (latched target)
ELSIF bTargetExtend AND NOT bSwitchExtended_eff THEN
    bOutSolenoidExtend  := TRUE;
    bOutSolenoidRetract := FALSE;

// CASE 2: Move to RETRACTED position (latched target)
ELSIF bTargetRetract AND NOT bSwitchRetracted_eff THEN
    bOutSolenoidRetract := TRUE;
    bOutSolenoidExtend  := FALSE;

// CASE 3: Target reached or no active target → stop both coils
ELSE
    bOutSolenoidExtend  := FALSE;
    bOutSolenoidRetract := FALSE;
END_IF;

(* ==========================================
   3. HMI STATUS FEEDBACK
   ========================================== *)
stHmi.bIsExtended        := bSwitchExtended_eff;
stHmi.bIsRetracted       := bSwitchRetracted_eff;
stHmi.bIsMoving          := bOutSolenoidExtend OR bOutSolenoidRetract;
stHmi.bOutSolenoidExtend  := bOutSolenoidExtend;
stHmi.bOutSolenoidRetract := bOutSolenoidRetract;

END_FUNCTION_BLOCK

// ---- POUs/PRG_IoMap.TcPOU
PROGRAM PRG_IoMap
VAR
END_VAR

ReadInputs();
WriteOutputs();

ACTION ReadInputs:
(* ==========================================
   READ INPUTS — copy raw GVL_IO.dIn[] channels into named GVL_App aliases.
   Each SOL-Spring actuator has both a Retracted and an Extended proximity
   switch (spring retracts, coil extends; both end positions get sensors).
   DI layout:
     dIn[1..2]   = SepSol1 (Retract, Extend)
     dIn[3..4]   = SepSol2 (Retract, Extend)
     dIn[5..6]   = SepSol3 (Retract, Extend)
     dIn[7..8]   = PushSol1 (Retract, Extend)
     dIn[9..10]  = PushSol2 (Retract, Extend)
     dIn[11..12] = PushSol3 (Retract, Extend)
     dIn[13]     = free (was Robot STAND_SEQ_DO; retired, comms are TCP-only)
     dIn[14..15] = GripSolL (Retract, Extend)
     dIn[16..17] = GripSolR (Retract, Extend)
     dIn[18]     = PlateSenL (plate-presence, left)
     dIn[19]     = PlateSenR (plate-presence, right)
     dIn[20]     = PB1 (grip in Manual / cycle-start bypass in Auto)
     dIn[21]     = PB2 (Sep jog in Manual)
     dIn[22]     = PB3 (Push jog in Manual)
     dIn[23..24] = free
   ========================================== *)
GVL_App.bSensorSepRetracted1  := GVL_IO.dIn[1];
GVL_App.bSensorSepExtended1   := GVL_IO.dIn[2];
GVL_App.bSensorSepRetracted2  := GVL_IO.dIn[3];
GVL_App.bSensorSepExtended2   := GVL_IO.dIn[4];
GVL_App.bSensorSepRetracted3  := GVL_IO.dIn[5];
GVL_App.bSensorSepExtended3   := GVL_IO.dIn[6];
GVL_App.bSensorPushRetracted1 := GVL_IO.dIn[7];
GVL_App.bSensorPushExtended1  := GVL_IO.dIn[8];
GVL_App.bSensorPushRetracted2 := GVL_IO.dIn[9];
GVL_App.bSensorPushExtended2  := GVL_IO.dIn[10];
GVL_App.bSensorPushRetracted3 := GVL_IO.dIn[11];
GVL_App.bSensorPushExtended3  := GVL_IO.dIn[12];

(* Grip pistons — DI 14..17. *)
GVL_App.bSensorGripRetractedL := GVL_IO.dIn[14];
GVL_App.bSensorGripExtendedL  := GVL_IO.dIn[15];
GVL_App.bSensorGripRetractedR := GVL_IO.dIn[16];
GVL_App.bSensorGripExtendedR  := GVL_IO.dIn[17];

(* Plate-presence sensors — DI 18..19. Both must be TRUE for WAIT_PLATE to
   advance the cycle into GRIP_EXTENDING. *)
GVL_App.bPlateSenL := GVL_IO.dIn[18];
GVL_App.bPlateSenR := GVL_IO.dIn[19];

(* Panel push buttons — DI 20..22. Consumer logic lives in MAIN (mode-gated
   jog OR cycle-start bypass). *)
GVL_App.bPb1 := GVL_IO.dIn[20];
GVL_App.bPb2 := GVL_IO.dIn[21];
GVL_App.bPb3 := GVL_IO.dIn[22];
END_ACTION

ACTION WriteOutputs:
(* ==========================================
   WRITE OUTPUTS — copy named GVL_App aliases into raw GVL_IO.dOut[] channels.
   Single Extend coil per actuator (SOL-Spring, spring retracts).
   DO layout:
     dOut[1..3]   = SepSol1..3 Extend coils
     dOut[4..6]   = PushSol1..3 Extend coils
     dOut[7]      = free (was PLC -> Robot STAND_SEQ_DI; retired, comms are TCP-only)
     dOut[8]      = GripSolL Extend coil
     dOut[9]      = GripSolR Extend coil
     dOut[10]     = LED1 (mirrors PB1)
     dOut[11]     = LED2 (mirrors PB2)
     dOut[12]     = LED3 (mirrors PB3)
     dOut[13..16] = free
   ========================================== *)
GVL_IO.dOut[1] := GVL_App.bValveSepExtend1;
GVL_IO.dOut[2] := GVL_App.bValveSepExtend2;
GVL_IO.dOut[3] := GVL_App.bValveSepExtend3;
GVL_IO.dOut[4] := GVL_App.bValvePushExtend1;
GVL_IO.dOut[5] := GVL_App.bValvePushExtend2;
GVL_IO.dOut[6] := GVL_App.bValvePushExtend3;

(* Grip piston extend coils. *)
GVL_IO.dOut[8] := GVL_App.bValveGripExtendL;
GVL_IO.dOut[9] := GVL_App.bValveGripExtendR;

(* Panel push-button status LEDs — mirror driven by MAIN. *)
GVL_IO.dOut[10] := GVL_App.bLedPb1;
GVL_IO.dOut[11] := GVL_App.bLedPb2;
GVL_IO.dOut[12] := GVL_App.bLedPb3;
END_ACTION

END_PROGRAM

// ---- GlobalTextList.TcGTLO
TEXTLIST GlobalTextList
  72 = '%s'
  899 = 'Auto'
  658 = 'Auto/Manual'
  841 = 'bManCmdExtend'
  294 = 'bManCmdRetract'
  296 = 'bManJogExtend'
  926 = 'bManJogRetract'
  57 = 'Man'
  58 = 'MOVING'
  429 = 'SimEXT'
  52 = 'SimRET'
END_TEXTLIST

// ---- VISUs/VISU_Home.TcVIS
VISUALIZATION VISU_Home  // 800x480
END_VISUALIZATION

// ---- VISUs/VISU_Piston.TcVIS
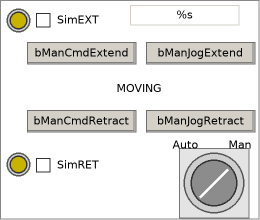
VISUALIZATION VISU_Piston  // 260x220
VAR_IN_OUT
	piston : ST_HmiPiston;
END_VAR
    Label (18,7 95x20)
    Textfield (130,5 109x20), "%s", text variable: piston.Name
    Button (146,42 109x22), "bManJogExtend"
        tap piston.bManJogExtend
    Button (146,110 109x22), "bManJogRetract"
        tap piston.bManJogRetract
    Button (27,110 109x22), "bManCmdRetract"
        tap piston.bManCmdRetract
    Button (27,42 109x22), "bManCmdExtend"
        tap piston.bManCmdExtend
    Checkbox (34,5 84x30), "SimEXT", variable: piston.bSimulateExtended
    Checkbox (34,150 84x30), "SimRET", variable: piston.bSimulateRetracted
    Lamp1 (4,7 29x27), variable: piston.bIsExtended, style: Lamp-Lamp1-Yellow
    Lamp1 (4,151 29x27), variable: piston.bIsRetracted, style: Lamp-Lamp1-Yellow
    Rectangle (0,-2 259x221)
    RotarySwitch (179,148 70x70), tooltip "Auto/Manual", variable: piston.bMode, behaviour: TOGGLE, style: Switch-RotarySwitch-Gray
    Label (167,135 37x20), "Auto", invisible if: NOT(piston.bMode)
    Label (220,135 40x20), "Man", invisible if: piston.bMode
    Label (86,77 106x23), "MOVING", invisible if: NOT(piston.bIsMoving)
END_VISUALIZATION

// ---- VISUs/VISU_Pistons.TcVIS
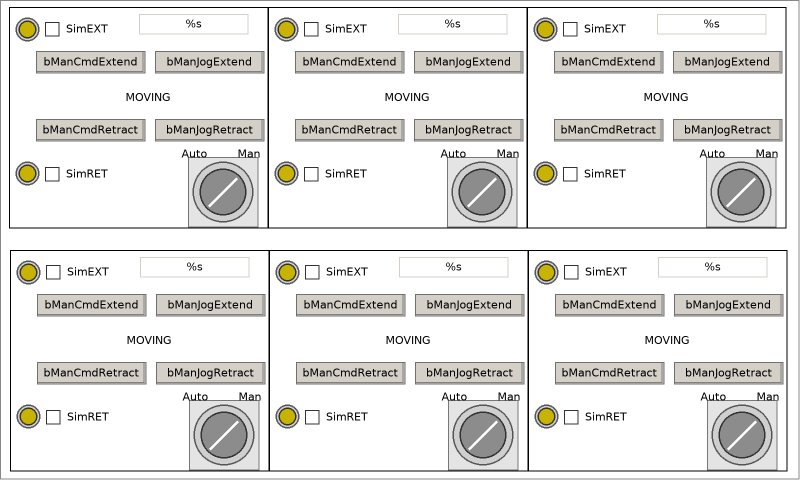
VISUALIZATION VISU_Pistons  // 800x480
    Frame (9,9 260x220)
        shows VISU_Piston(piston := GVL_HMI.stSepSol1)
    Frame (10,252 260x220)
        shows VISU_Piston(piston := GVL_HMI.stPushSol1)
    Frame (268,9 260x220)
        shows VISU_Piston(piston := GVL_HMI.stSepSol2)
    Frame (269,252 260x220)
        shows VISU_Piston(piston := GVL_HMI.stPushSol2)
    Frame (527,9 260x220)
        shows VISU_Piston(piston := GVL_HMI.stSepSol3)
    Frame (528,252 260x220)
        shows VISU_Piston(piston := GVL_HMI.stPushSol3)
END_VISUALIZATION

// ---- VISUs/VISU_Robot.TcVIS
VISUALIZATION VISU_Robot  // 800x480
END_VISUALIZATION

// ---- VISUs/VISU_AutoCycle.TcVIS
VISUALIZATION VISU_AutoCycle  // 800x480
END_VISUALIZATION

// ---- VISUs/VISU_Diagnostics.TcVIS
VISUALIZATION VISU_Diagnostics  // 800x480
END_VISUALIZATION
